LIN {X 0,Y 506.192,Z 351.476,A -85,B 0,C 180,E1 -5678.842,E2 -5678.842} C_VEL
LIN {X 0,Y 505.573,Z 365.781,A -85,B 0,C 180,E1 -5679.704,E2 -5679.704} C_VEL
LIN {X 0,Y 505.041,Z 378.228,A -85,B 0,C 180,E1 -5680.625,E2 -5680.625} C_VEL
LIN {X 0,Y 504.462,Z 389.865,A -85,B 0,C 180,E1 -5681.655,E2 -5681.655} C_VEL
LIN {X 0,Y 503.901,Z 401.554,A -85,B 0,C 180,E1 -5682.894,E2 -5682.894} C_VEL
LIN {X 0,Y 503.396,Z 411.462,A -85,B 0,C 180,E1 -5684.142,E2 -5684.142} C_VEL
LIN {X 0,Y 502.965,Z 421.023,A -85,B 0,C 180,E1 -5685.583,E2 -5685.583} C_VEL
LIN {X 0,Y 502.631,Z 429.216,A -85,B 0,C 180,E1 -5687.075,E2 -5687.075} C_VEL
LIN {X 0,Y 502.473,Z 434.837,A -85,B 0,C 180,E1 -5688.301,E2 -5688.301} C_VEL
LIN {X 0,Y 502.272,Z 441.149,A -85,B 0,C 180,E1 -5689.99,E2 -5689.99} C_VEL
LIN {X 0,Y 502.192,Z 445.104,A -85,B 0,C 180,E1 -5691.338,E2 -5691.338} C_VEL
LIN {X 0,Y 502.044,Z 448.907,A -85,B 0,C 180,E1 -5693.077,E2 -5693.077} C_VEL
LIN {X 0,Y 501.982,Z 451.304,A -85,B 0,C 180,E1 -5694.836,E2 -5694.836} C_VEL
LIN {X 0,Y 501.984,Z 452.341,A -85,B 0,C 180,E1 -5696.616,E2 -5696.616} C_VEL
LIN {X 0,Y 501.997,Z 451.979,A -85,B 0,C 180,E1 -5698.425,E2 -5698.425} C_VEL
LIN {X 0,Y 502.054,Z 450.118,A -85,B 0,C 180,E1 -5700.261,E2 -5700.261} C_VEL
LIN {X 0,Y 502.066,Z 448.297,A -85,B 0,C 180,E1 -5701.362,E2 -5701.362} C_VEL
LIN {X 0,Y 502.167,Z 444.274,A -85,B 0,C 180,E1 -5703.081,E2 -5703.081} C_VEL
LIN {X 0,Y 502.321,Z 439.329,A -85,B 0,C 180,E1 -5704.647,E2 -5704.647} C_VEL
LIN {X 0,Y 502.482,Z 433.012,A -85,B 0,C 180,E1 -5706.223,E2 -5706.223} C_VEL
LIN {X 0,Y 502.787,Z 425.506,A -85,B 0,C 180,E1 -5707.736,E2 -5707.736} C_VEL
LIN {X 0,Y 503.138,Z 416.684,A -85,B 0,C 180,E1 -5709.203,E2 -5709.203} C_VEL
LIN {X 0,Y 503.572,Z 407.62,A -85,B 0,C 180,E1 -5710.464,E2 -5710.464} C_VEL
LIN {X 0,Y 504.123,Z 396.604,A -85,B 0,C 180,E1 -5711.756,E2 -5711.756} C_VEL
LIN {X 0,Y 504.628,Z 385.523,A -85,B 0,C 180,E1 -5712.848,E2 -5712.848} C_VEL
LIN {X 0,Y 505.24,Z 373.889,A -85,B 0,C 180,E1 -5713.811,E2 -5713.811} C_VEL
LIN {X 0,Y 505.78,Z 361.268,A -85,B 0,C 180,E1 -5714.683,E2 -5714.683} C_VEL
LIN {X 0,Y 506.347,Z 346.906,A -85,B 0,C 180,E1 -5715.486,E2 -5715.486} C_VEL
LIN {X 0,Y 506.899,Z 331.848,A -85,B 0,C 180,E1 -5716.134,E2 -5716.134} C_VEL
LIN {X 0,Y 507.236,Z 316.604,A -85,B 0,C 180,E1 -5716.616,E2 -5716.616} C_VEL
LIN {X 0,Y 507.491,Z 300.362,A -85,B 0,C 180,E1 -5716.947,E2 -5716.947} C_VEL
LIN {X 0,Y 508.749,Z 153.983,A -85,B 0,C 180,E1 -5719.077,E2 -5719.077} C_VEL
LIN {X 0,Y 506.279,Z 139.939,A -85,B 0,C 180,E1 -5719.421,E2 -5719.421} C_VEL
LIN {X 0,Y 506.545,Z 123.358,A -85,B 0,C 180,E1 -5721.177,E2 -5721.177} C_VEL
LIN {X 0,Y 502.795,Z 108.482,A -85,B 0,C 180,E1 -5722.971,E2 -5722.971} C_VEL
LIN {X 0,Y 502.806,Z 108.482,A -85,B 0,C 180,E1 -5726.006,E2 -5726.006} C_VEL
LIN {X 0,Y 502.799,Z 108.477,A -85,B 0,C 180,E1 -5728.857,E2 -5728.857} C_VEL
LIN {X 0,Y 502.847,Z 108.477,A -85,B 0,C 180,E1 -5731.705,E2 -5731.705} C_VEL
LIN {X 0,Y 502.843,Z 108.473,A -85,B 0,C 180,E1 -5734.324,E2 -5734.324} C_VEL
LIN {X 0,Y 502.818,Z 108.529,A -85,B 0,C 180,E1 -5736.986,E2 -5736.986} C_VEL
LIN {X 0,Y 503.872,Z 112.951,A -85,B 0,C 180,E1 -5737.604,E2 -5737.604} C_VEL
LIN {X 0,Y 508.613,Z 125.414,A -85,B 0,C 180,E1 -5738.027,E2 -5738.027} C_VEL
LIN {X 0,Y 507.559,Z 222.564,A -85,B 0,C 180,E1 -5739.562,E2 -5739.562} C_VEL
LIN {X 0,Y 506.94,Z 279.945,A -85,B 0,C 180,E1 -5740.465,E2 -5740.465} C_VEL
LIN {X 0,Y 506.668,Z 295.372,A -85,B 0,C 180,E1 -5740.872,E2 -5740.872} C_VEL
LIN {X 0,Y 506.263,Z 310.367,A -85,B 0,C 180,E1 -5741.432,E2 -5741.432} C_VEL
LIN {X 0,Y 505.837,Z 324.005,A -85,B 0,C 180,E1 -5742.097,E2 -5742.097} C_VEL
LIN {X 0,Y 505.288,Z 337.428,A -85,B 0,C 180,E1 -5742.913,E2 -5742.913} C_VEL
LIN {X 0,Y 504.764,Z 350.501,A -85,B 0,C 180,E1 -5743.886,E2 -5743.886} C_VEL
LIN {X 0,Y 504.241,Z 363.457,A -85,B 0,C 180,E1 -5745.057,E2 -5745.057} C_VEL
LIN {X 0,Y 503.727,Z 374.703,A -85,B 0,C 180,E1 -5746.279,E2 -5746.279} C_VEL
LIN {X 0,Y 503.243,Z 385.732,A -85,B 0,C 180,E1 -5747.724,E2 -5747.724} C_VEL
LIN {X 0,Y 502.954,Z 394.624,A -85,B 0,C 180,E1 -5749.126,E2 -5749.126} C_VEL
LIN {X 0,Y 502.597,Z 403.052,A -85,B 0,C 180,E1 -5750.746,E2 -5750.746} C_VEL
LIN {X 0,Y 502.405,Z 409.809,A -85,B 0,C 180,E1 -5752.363,E2 -5752.363} C_VEL
LIN {X 0,Y 502.315,Z 415.092,A -85,B 0,C 180,E1 -5753.976,E2 -5753.976} C_VEL
LIN {X 0,Y 502.12,Z 418.131,A -85,B 0,C 180,E1 -5755.182,E2 -5755.182} C_VEL
LIN {X 0,Y 502.231,Z 421.123,A -85,B 0,C 180,E1 -5756.791,E2 -5756.791} C_VEL
LIN {X 0,Y 502.036,Z 422.952,A -85,B 0,C 180,E1 -5758.395,E2 -5758.395} C_VEL
LIN {X 0,Y 502.002,Z 423.613,A -85,B 0,C 180,E1 -5760,E2 -5760} C_VEL
LIN {X 0,Y 502.038,Z 423.077,A -85,B 0,C 180,E1 -5761.604,E2 -5761.604} C_VEL
LIN {X 0,Y 502.249,Z 421.385,A -85,B 0,C 180,E1 -5763.208,E2 -5763.208} C_VEL
LIN {X 0,Y 502.141,Z 418.525,A -85,B 0,C 180,E1 -5764.817,E2 -5764.817} C_VEL
LIN {X 0,Y 502.333,Z 414.388,A -85,B 0,C 180,E1 -5766.426,E2 -5766.426} C_VEL
LIN {X 0,Y 502.462,Z 408.89,A -85,B 0,C 180,E1 -5768.04,E2 -5768.04} C_VEL
LIN {X 0,Y 502.666,Z 401.854,A -85,B 0,C 180,E1 -5769.658,E2 -5769.658} C_VEL
LIN {X 0,Y 503.001,Z 394.271,A -85,B 0,C 180,E1 -5771.076,E2 -5771.076} C_VEL
LIN {X 0,Y 503.278,Z 385.393,A -85,B 0,C 180,E1 -5772.459,E2 -5772.459} C_VEL
LIN {X 0,Y 503.727,Z 375.704,A -85,B 0,C 180,E1 -5773.72,E2 -5773.72} C_VEL
LIN {X 0,Y 504.195,Z 364.498,A -85,B 0,C 180,E1 -5774.944,E2 -5774.944} C_VEL
LIN {X 0,Y 504.763,Z 351.596,A -85,B 0,C 180,E1 -5776.113,E2 -5776.113} C_VEL
LIN {X 0,Y 505.237,Z 338.543,A -85,B 0,C 180,E1 -5777.089,E2 -5777.089} C_VEL
LIN {X 0,Y 505.762,Z 325.103,A -85,B 0,C 180,E1 -5777.905,E2 -5777.905} C_VEL
LIN {X 0,Y 506.147,Z 311.424,A -85,B 0,C 180,E1 -5778.572,E2 -5778.572} C_VEL
LIN {X 0,Y 506.518,Z 296.117,A -85,B 0,C 180,E1 -5779.142,E2 -5779.142} C_VEL
LIN {X 0,Y 506.766,Z 280.632,A -85,B 0,C 180,E1 -5779.546,E2 -5779.546} C_VEL
LIN {X 0,Y 508.512,Z 155.31,A -85,B 0,C 180,E1 -5781.608,E2 -5781.608} C_VEL
LIN {X 0,Y 508.849,Z 129.1,A -85,B 0,C 180,E1 -5782.07,E2 -5782.07} C_VEL
LIN {X 0,Y 506.949,Z 122.35,A -85,B 0,C 180,E1 -5782.298,E2 -5782.298} C_VEL
LIN {X 0,Y 504.919,Z 117.566,A -85,B 0,C 180,E1 -5782.524,E2 -5782.524} C_VEL
LIN {X 0,Y 502.798,Z 108.482,A -85,B 0,C 180,E1 -5784.394,E2 -5784.394} C_VEL
LIN {X 0,Y 502.79,Z 108.484,A -85,B 0,C 180,E1 -5787.469,E2 -5787.469} C_VEL
LIN {X 0,Y 502.802,Z 108.48,A -85,B 0,C 180,E1 -5790.211,E2 -5790.211} C_VEL
LIN {X 0,Y 502.802,Z 108.48,A -85,B 0,C 180,E1 -5793.033,E2 -5793.033} C_VEL
LIN {X 0,Y 502.766,Z 108.485,A -85,B 0,C 180,E1 -5795.952,E2 -5795.952} C_VEL
LIN {X 0,Y 502.795,Z 108.481,A -85,B 0,C 180,E1 -5798.976,E2 -5798.976} C_VEL
LIN {X 0,Y 502.743,Z 108.484,A -85,B 0,C 180,E1 -5802.192,E2 -5802.192} C_VEL
LIN {X 0,Y 502.784,Z 108.483,A -85,B 0,C 180,E1 -5805.47,E2 -5805.47} C_VEL
LIN {X 0,Y 502.763,Z 108.487,A -85,B 0,C 180,E1 -5808.928,E2 -5808.928} C_VEL
LIN {X 0,Y 502.788,Z 108.479,A -85,B 0,C 180,E1 -5812.046,E2 -5812.046} C_VEL
LIN {X 0,Y 502.786,Z 108.485,A -85,B 0,C 180,E1 -5815.033,E2 -5815.033} C_VEL
LIN {X 0,Y 502.771,Z 108.484,A -85,B 0,C 180,E1 -5817.914,E2 -5817.914} C_VEL
LIN {X 0,Y 502.802,Z 108.672,A -85,B 0,C 180,E1 -5819.834,E2 -5819.834} C_VEL
LIN {X 0,Y 505.92,Z 121.058,A -85,B 0,C 180,E1 -5821.816,E2 -5821.816} C_VEL
LIN {X 0,Y 506.557,Z 124.311,A -85,B 0,C 180,E1 -5822.304,E2 -5822.304} C_VEL
LIN {X 0,Y 505.722,Z 144.394,A -85,B 0,C 180,E1 -5824.967,E2 -5824.967} C_VEL
LIN {X 0,Y 504.954,Z 164.114,A -85,B 0,C 180,E1 -5827.496,E2 -5827.496} C_VEL
LIN {X 0,Y 508.497,Z 185.654,A -85,B 0,C 180,E1 -5828.073,E2 -5828.073} C_VEL
LIN {X 0,Y 507.022,Z 292.758,A -85,B 0,C 180,E1 -5829.83,E2 -5829.83} C_VEL
LIN {X 0,Y 506.548,Z 333.914,A -85,B 0,C 180,E1 -5830.497,E2 -5830.497} C_VEL
LIN {X 0,Y 506.136,Z 349.417,A -85,B 0,C 180,E1 -5830.905,E2 -5830.905} C_VEL
LIN {X 0,Y 505.713,Z 364.455,A -85,B 0,C 180,E1 -5831.464,E2 -5831.464} C_VEL
LIN {X 0,Y 505.165,Z 379.158,A -85,B 0,C 180,E1 -5832.177,E2 -5832.177} C_VEL
LIN {X 0,Y 504.657,Z 392.632,A -85,B 0,C 180,E1 -5832.995,E2 -5832.995} C_VEL
LIN {X 0,Y 504.186,Z 406.022,A -85,B 0,C 180,E1 -5833.987,E2 -5833.987} C_VEL
LIN {X 0,Y 503.687,Z 417.91,A -85,B 0,C 180,E1 -5835.041,E2 -5835.041} C_VEL
LIN {X 0,Y 503.287,Z 429.5,A -85,B 0,C 180,E1 -5836.267,E2 -5836.267} C_VEL
LIN {X 0,Y 502.932,Z 439.231,A -85,B 0,C 180,E1 -5837.491,E2 -5837.491} C_VEL
LIN {X 0,Y 502.691,Z 447.494,A -85,B 0,C 180,E1 -5838.713,E2 -5838.713} C_VEL
LIN {X 0,Y 502.423,Z 455.624,A -85,B 0,C 180,E1 -5840.133,E2 -5840.133} C_VEL
LIN {X 0,Y 502.285,Z 462.353,A -85,B 0,C 180,E1 -5841.552,E2 -5841.552} C_VEL
LIN {X 0,Y 502.221,Z 468.522,A -85,B 0,C 180,E1 -5843.169,E2 -5843.169} C_VEL
LIN {X 0,Y 502.146,Z 473.251,A -85,B 0,C 180,E1 -5844.78,E2 -5844.78} C_VEL
LIN {X 0,Y 502.13,Z 475.867,A -85,B 0,C 180,E1 -5845.987,E2 -5845.987} C_VEL
LIN {X 0,Y 502.117,Z 478.31,A -85,B 0,C 180,E1 -5847.593,E2 -5847.593} C_VEL
LIN {X 0,Y 501.993,Z 479.548,A -85,B 0,C 180,E1 -5849.198,E2 -5849.198} C_VEL
LIN {X 0,Y 501.992,Z 479.577,A -85,B 0,C 180,E1 -5850.802,E2 -5850.802} C_VEL
LIN {X 0,Y 502.117,Z 478.396,A -85,B 0,C 180,E1 -5852.407,E2 -5852.407} C_VEL
LIN {X 0,Y 502.129,Z 476.018,A -85,B 0,C 180,E1 -5854.013,E2 -5854.013} C_VEL
LIN {X 0,Y 502.195,Z 472.398,A -85,B 0,C 180,E1 -5855.622,E2 -5855.622} C_VEL
LIN {X 0,Y 502.234,Z 467.436,A -85,B 0,C 180,E1 -5857.235,E2 -5857.235} C_VEL
LIN {X 0,Y 502.313,Z 461,A -85,B 0,C 180,E1 -5858.853,E2 -5858.853} C_VEL
LIN {X 0,Y 502.584,Z 452.92,A -85,B 0,C 180,E1 -5860.474,E2 -5860.474} C_VEL
LIN {X 0,Y 502.804,Z 444.129,A -85,B 0,C 180,E1 -5861.922,E2 -5861.922} C_VEL
LIN {X 0,Y 503.195,Z 433.884,A -85,B 0,C 180,E1 -5863.324,E2 -5863.324} C_VEL
LIN {X 0,Y 503.616,Z 423.234,A -85,B 0,C 180,E1 -5864.548,E2 -5864.548} C_VEL
LIN {X 0,Y 504.109,Z 410.905,A -85,B 0,C 180,E1 -5865.736,E2 -5865.736} C_VEL
LIN {X 0,Y 504.603,Z 399.061,A -85,B 0,C 180,E1 -5866.694,E2 -5866.694} C_VEL
LIN {X 0,Y 505.206,Z 385.293,A -85,B 0,C 180,E1 -5867.612,E2 -5867.612} C_VEL
LIN {X 0,Y 505.75,Z 371.064,A -85,B 0,C 180,E1 -5868.377,E2 -5868.377} C_VEL
LIN {X 0,Y 506.262,Z 356.646,A -85,B 0,C 180,E1 -5868.982,E2 -5868.982} C_VEL
LIN {X 0,Y 506.665,Z 341.674,A -85,B 0,C 180,E1 -5869.445,E2 -5869.445} C_VEL
LIN {X 0,Y 506.929,Z 325.194,A -85,B 0,C 180,E1 -5869.777,E2 -5869.777} C_VEL
LIN {X 0,Y 508.535,Z 184.49,A -85,B 0,C 180,E1 -5871.962,E2 -5871.962} C_VEL
LIN {X 0,Y 508.192,Z 179.447,A -85,B 0,C 180,E1 -5872.061,E2 -5872.061} C_VEL
LIN {X 0,Y 506.015,Z 165.025,A -85,B 0,C 180,E1 -5872.411,E2 -5872.411} C_VEL
LIN {X 0,Y 506.86,Z 142.117,A -85,B 0,C 180,E1 -5874.69,E2 -5874.69} C_VEL
LIN {X 0,Y 507.529,Z 126.06,A -85,B 0,C 180,E1 -5876.303,E2 -5876.303} C_VEL
LIN {X 0,Y 502.788,Z 108.483,A -85,B 0,C 180,E1 -5878.404,E2 -5878.404} C_VEL
LIN {X 0,Y 502.785,Z 108.484,A -85,B 0,C 180,E1 -5881.144,E2 -5881.144} C_VEL
LIN {X 0,Y 502.785,Z 108.478,A -85,B 0,C 180,E1 -5883.995,E2 -5883.995} C_VEL
LIN {X 0,Y 502.763,Z 108.486,A -85,B 0,C 180,E1 -5887.176,E2 -5887.176} C_VEL
LIN {X 0,Y 502.77,Z 108.481,A -85,B 0,C 180,E1 -5890.017,E2 -5890.017} C_VEL
LIN {X 0,Y 502.746,Z 108.484,A -85,B 0,C 180,E1 -5893.234,E2 -5893.234} C_VEL
LIN {X 0,Y 502.777,Z 108.476,A -85,B 0,C 180,E1 -5895.66,E2 -5895.66} C_VEL
LIN {X 0,Y 502.764,Z 108.483,A -85,B 0,C 180,E1 -5899.012,E2 -5899.012} C_VEL
LIN {X 0,Y 502.789,Z 108.48,A -85,B 0,C 180,E1 -5902.046,E2 -5902.046} C_VEL
LIN {X 0,Y 502.791,Z 108.48,A -85,B 0,C 180,E1 -5905.034,E2 -5905.034} C_VEL
LIN {X 0,Y 502.781,Z 108.482,A -85,B 0,C 180,E1 -5907.915,E2 -5907.915} C_VEL
LIN {X 0,Y 502.804,Z 108.481,A -85,B 0,C 180,E1 -5910.711,E2 -5910.711} C_VEL
LIN {X 0,Y 502.774,Z 108.482,A -85,B 0,C 180,E1 -5913.46,E2 -5913.46} C_VEL
LIN {X 0,Y 502.786,Z 108.557,A -85,B 0,C 180,E1 -5916.387,E2 -5916.387} C_VEL
LIN {X 0,Y 504.707,Z 116.182,A -85,B 0,C 180,E1 -5917.588,E2 -5917.588} C_VEL
LIN {X 0,Y 507.891,Z 125.008,A -85,B 0,C 180,E1 -5917.921,E2 -5917.921} C_VEL
LIN {X 0,Y 508.835,Z 129.707,A -85,B 0,C 180,E1 -5918.056,E2 -5918.056} C_VEL
LIN {X 0,Y 507.257,Z 231.397,A -85,B 0,C 180,E1 -5919.761,E2 -5919.761} C_VEL
LIN {X 0,Y 506.727,Z 280.59,A -85,B 0,C 180,E1 -5920.557,E2 -5920.557} C_VEL
LIN {X 0,Y 506.476,Z 295.923,A -85,B 0,C 180,E1 -5920.956,E2 -5920.956} C_VEL
LIN {X 0,Y 506.123,Z 310.178,A -85,B 0,C 180,E1 -5921.48,E2 -5921.48} C_VEL
LIN {X 0,Y 505.757,Z 323.108,A -85,B 0,C 180,E1 -5922.095,E2 -5922.095} C_VEL
LIN {X 0,Y 505.238,Z 336.924,A -85,B 0,C 180,E1 -5922.911,E2 -5922.911} C_VEL
LIN {X 0,Y 504.732,Z 350.42,A -85,B 0,C 180,E1 -5923.898,E2 -5923.898} C_VEL
LIN {X 0,Y 504.25,Z 362.346,A -85,B 0,C 180,E1 -5924.955,E2 -5924.955} C_VEL
LIN {X 0,Y 503.807,Z 373.008,A -85,B 0,C 180,E1 -5926.076,E2 -5926.076} C_VEL
LIN {X 0,Y 503.419,Z 382.834,A -85,B 0,C 180,E1 -5927.299,E2 -5927.299} C_VEL
LIN {X 0,Y 503.038,Z 392.387,A -85,B 0,C 180,E1 -5928.721,E2 -5928.721} C_VEL
LIN {X 0,Y 502.689,Z 400.304,A -85,B 0,C 180,E1 -5930.139,E2 -5930.139} C_VEL
LIN {X 0,Y 502.515,Z 406.842,A -85,B 0,C 180,E1 -5931.556,E2 -5931.556} C_VEL
LIN {X 0,Y 502.311,Z 412.936,A -85,B 0,C 180,E1 -5933.21,E2 -5933.21} C_VEL
LIN {X 0,Y 502.275,Z 416.298,A -85,B 0,C 180,E1 -5934.379,E2 -5934.379} C_VEL
LIN {X 0,Y 502.189,Z 419.867,A -85,B 0,C 180,E1 -5935.988,E2 -5935.988} C_VEL
LIN {X 0,Y 502.13,Z 422.215,A -85,B 0,C 180,E1 -5937.594,E2 -5937.594} C_VEL
LIN {X 0,Y 502.003,Z 423.399,A -85,B 0,C 180,E1 -5939.198,E2 -5939.198} C_VEL
LIN {X 0,Y 502.003,Z 423.386,A -85,B 0,C 180,E1 -5940.802,E2 -5940.802} C_VEL
LIN {X 0,Y 502.131,Z 422.213,A -85,B 0,C 180,E1 -5942.407,E2 -5942.407} C_VEL
LIN {X 0,Y 502.188,Z 419.88,A -85,B 0,C 180,E1 -5944.013,E2 -5944.013} C_VEL
LIN {X 0,Y 502.267,Z 416.329,A -85,B 0,C 180,E1 -5945.621,E2 -5945.621} C_VEL
LIN {X 0,Y 502.361,Z 411.477,A -85,B 0,C 180,E1 -5947.234,E2 -5947.234} C_VEL
LIN {X 0,Y 502.508,Z 405.194,A -85,B 0,C 180,E1 -5948.85,E2 -5948.85} C_VEL
LIN {X 0,Y 502.772,Z 397.283,A -85,B 0,C 180,E1 -5950.47,E2 -5950.47} C_VEL
LIN {X 0,Y 503.038,Z 388.849,A -85,B 0,C 180,E1 -5951.887,E2 -5951.887} C_VEL
LIN {X 0,Y 503.54,Z 378.594,A -85,B 0,C 180,E1 -5953.315,E2 -5953.315} C_VEL
LIN {X 0,Y 504.008,Z 368.103,A -85,B 0,C 180,E1 -5954.537,E2 -5954.537} C_VEL
LIN {X 0,Y 504.5,Z 356.654,A -85,B 0,C 180,E1 -5955.66,E2 -5955.66} C_VEL
LIN {X 0,Y 505.013,Z 344.225,A -85,B 0,C 180,E1 -5956.68,E2 -5956.68} C_VEL
LIN {X 0,Y 505.543,Z 330.609,A -85,B 0,C 180,E1 -5957.6,E2 -5957.6} C_VEL
LIN {X 0,Y 506.037,Z 316.494,A -85,B 0,C 180,E1 -5958.367,E2 -5958.367} C_VEL
LIN {X 0,Y 506.511,Z 300.879,A -85,B 0,C 180,E1 -5959.02,E2 -5959.02} C_VEL
LIN {X 0,Y 506.843,Z 285.314,A -85,B 0,C 180,E1 -5959.491,E2 -5959.491} C_VEL
LIN {X 0,Y 507.044,Z 269.676,A -85,B 0,C 180,E1 -5959.799,E2 -5959.799} C_VEL
LIN {X 0,Y 508.646,Z 129.723,A -85,B 0,C 180,E1 -5961.977,E2 -5961.977} C_VEL
LIN {X 0,Y 506.606,Z 120.903,A -85,B 0,C 180,E1 -5962.212,E2 -5962.212} C_VEL
LIN {X 0,Y 503.925,Z 113.653,A -85,B 0,C 180,E1 -5962.479,E2 -5962.479} C_VEL
LIN {X 0,Y 502.805,Z 108.48,A -85,B 0,C 180,E1 -5963.367,E2 -5963.367} C_VEL
LIN {X 0,Y 502.814,Z 108.475,A -85,B 0,C 180,E1 -5966.569,E2 -5966.569} C_VEL
LIN {X 0,Y 502.812,Z 108.48,A -85,B 0,C 180,E1 -5969.934,E2 -5969.934} C_VEL
LIN {X 0,Y 502.804,Z 108.477,A -85,B 0,C 180,E1 -5973.034,E2 -5973.034} C_VEL
LIN {X 0,Y 502.77,Z 108.483,A -85,B 0,C 180,E1 -5975.888,E2 -5975.888} C_VEL
LIN {X 0,Y 502.096,Z 108.564,A -85,B 0,C 180,E1 -5976.556,E2 -5976.556} C_VEL
LIN {X 0,Y 499.241,Z 108.925,A -85,B 0,C 180,E1 -5977.64,E2 -5977.64} C_VEL
LIN {X 0,Y 496.837,Z 109.22,A -85,B 0,C 180,E1 -5978.514,E2 -5978.514} C_VEL
LIN {X 0,Y 495.816,Z 109.349,A -85,B 0,C 180,E1 -5979.189,E2 -5979.189} C_VEL
LIN {X 0,Y 495.738,Z 109.358,A -85,B 0,C 180,E1 -5979.417,E2 -5979.417} C_VEL
LIN {X 0,Y 495.714,Z 109.358,A -85,B 0,C 180,E1 -5982.504,E2 -5982.504} C_VEL
LIN {X 0,Y 495.739,Z 109.355,A -85,B 0,C 180,E1 -5985.141,E2 -5985.141} C_VEL
LIN {X 0,Y 495.726,Z 109.351,A -85,B 0,C 180,E1 -5988.216,E2 -5988.216} C_VEL
LIN {X 0,Y 495.748,Z 109.357,A -85,B 0,C 180,E1 -5991.408,E2 -5991.408} C_VEL
LIN {X 0,Y 495.745,Z 109.346,A -85,B 0,C 180,E1 -5994.462,E2 -5994.462} C_VEL
LIN {X 0,Y 495.753,Z 109.356,A -85,B 0,C 180,E1 -5997.404,E2 -5997.404} C_VEL
LIN {X 0,Y 495.742,Z 109.35,A -85,B 0,C 180,E1 -6000.252,E2 -6000.252} C_VEL
LIN {X 0,Y 495.742,Z 109.357,A -85,B 0,C 180,E1 -6003.271,E2 -6003.271} C_VEL
LIN {X 0,Y 495.737,Z 109.355,A -85,B 0,C 180,E1 -6006.612,E2 -6006.612} C_VEL
LIN {X 0,Y 495.782,Z 109.348,A -85,B 0,C 180,E1 -6009.324,E2 -6009.324} C_VEL
LIN {X 0,Y 495.764,Z 109.352,A -85,B 0,C 180,E1 -6011.828,E2 -6011.828} C_VEL
LIN {X 0,Y 495.777,Z 109.352,A -85,B 0,C 180,E1 -6015.217,E2 -6015.217} C_VEL
LIN {X 0,Y 495.854,Z 109.346,A -85,B 0,C 180,E1 -6018.555,E2 -6018.555} C_VEL
LIN {X 0,Y 495.814,Z 109.348,A -85,B 0,C 180,E1 -6021.851,E2 -6021.851} C_VEL
LIN {X 0,Y 495.819,Z 109.347,A -85,B 0,C 180,E1 -6025.121,E2 -6025.121} C_VEL
LIN {X 0,Y 495.977,Z 109.33,A -85,B 0,C 180,E1 -6027.564,E2 -6027.564} C_VEL
LIN {X 0,Y 495.904,Z 109.404,A -85,B 0,C 180,E1 -6029.746,E2 -6029.746} C_VEL
LIN {X 0,Y 498.874,Z 123.212,A -85,B 0,C 180,E1 -6031.816,E2 -6031.816} C_VEL
LIN {X 0,Y 498.743,Z 134.952,A -85,B 0,C 180,E1 -6033.433,E2 -6033.433} C_VEL
LIN {X 0,Y 498.575,Z 141.915,A -85,B 0,C 180,E1 -6034.36,E2 -6034.36} C_VEL
LIN {X 0,Y 502.108,Z 158.195,A -85,B 0,C 180,E1 -6034.776,E2 -6034.776} C_VEL
LIN {X 0,Y 500.735,Z 307.945,A -85,B 0,C 180,E1 -6037.004,E2 -6037.004} C_VEL
LIN {X 0,Y 500.429,Z 323.034,A -85,B 0,C 180,E1 -6037.388,E2 -6037.388} C_VEL
LIN {X 0,Y 499.964,Z 337.824,A -85,B 0,C 180,E1 -6037.928,E2 -6037.928} C_VEL
LIN {X 0,Y 499.425,Z 351.76,A -85,B 0,C 180,E1 -6038.599,E2 -6038.599} C_VEL
LIN {X 0,Y 498.832,Z 364.756,A -85,B 0,C 180,E1 -6039.381,E2 -6039.381} C_VEL
LIN {X 0,Y 498.254,Z 377.945,A -85,B 0,C 180,E1 -6040.361,E2 -6040.361} C_VEL
LIN {X 0,Y 497.581,Z 389.69,A -85,B 0,C 180,E1 -6041.405,E2 -6041.405} C_VEL
LIN {X 0,Y 496.995,Z 401.325,A -85,B 0,C 180,E1 -6042.648,E2 -6042.648} C_VEL
LIN {X 0,Y 496.464,Z 411.384,A -85,B 0,C 180,E1 -6043.925,E2 -6043.925} C_VEL
LIN {X 0,Y 495.961,Z 420.964,A -85,B 0,C 180,E1 -6045.381,E2 -6045.381} C_VEL
LIN {X 0,Y 495.606,Z 429.237,A -85,B 0,C 180,E1 -6046.9,E2 -6046.9} C_VEL
LIN {X 0,Y 495.439,Z 435.041,A -85,B 0,C 180,E1 -6048.185,E2 -6048.185} C_VEL
LIN {X 0,Y 495.213,Z 441.414,A -85,B 0,C 180,E1 -6049.914,E2 -6049.914} C_VEL
LIN {X 0,Y 495.073,Z 446.303,A -85,B 0,C 180,E1 -6051.66,E2 -6051.66} C_VEL
LIN {X 0,Y 494.924,Z 449.786,A -85,B 0,C 180,E1 -6053.429,E2 -6053.429} C_VEL
LIN {X 0,Y 494.866,Z 451.874,A -85,B 0,C 180,E1 -6055.217,E2 -6055.217} C_VEL
LIN {X 0,Y 494.886,Z 452.604,A -85,B 0,C 180,E1 -6057.029,E2 -6057.029} C_VEL
LIN {X 0,Y 494.914,Z 451.885,A -85,B 0,C 180,E1 -6058.869,E2 -6058.869} C_VEL
LIN {X 0,Y 494.954,Z 450.732,A -85,B 0,C 180,E1 -6059.984,E2 -6059.984} C_VEL
LIN {X 0,Y 495,Z 447.939,A -85,B 0,C 180,E1 -6061.69,E2 -6061.69} C_VEL
LIN {X 0,Y 495.089,Z 444.599,A -85,B 0,C 180,E1 -6063.119,E2 -6063.119} C_VEL
LIN {X 0,Y 495.238,Z 440.025,A -85,B 0,C 180,E1 -6064.604,E2 -6064.604} C_VEL
LIN {X 0,Y 495.425,Z 433.546,A -85,B 0,C 180,E1 -6066.27,E2 -6066.27} C_VEL
LIN {X 0,Y 495.763,Z 426.061,A -85,B 0,C 180,E1 -6067.815,E2 -6067.815} C_VEL
LIN {X 0,Y 496.148,Z 416.844,A -85,B 0,C 180,E1 -6069.379,E2 -6069.379} C_VEL
LIN {X 0,Y 496.627,Z 408.089,A -85,B 0,C 180,E1 -6070.615,E2 -6070.615} C_VEL
LIN {X 0,Y 497.193,Z 397.305,A -85,B 0,C 180,E1 -6071.905,E2 -6071.905} C_VEL
LIN {X 0,Y 497.73,Z 386.135,A -85,B 0,C 180,E1 -6073.029,E2 -6073.029} C_VEL
LIN {X 0,Y 498.398,Z 374.453,A -85,B 0,C 180,E1 -6074.014,E2 -6074.014} C_VEL
LIN {X 0,Y 498.967,Z 361.909,A -85,B 0,C 180,E1 -6074.899,E2 -6074.899} C_VEL
LIN {X 0,Y 499.556,Z 348.544,A -85,B 0,C 180,E1 -6075.667,E2 -6075.667} C_VEL
LIN {X 0,Y 500.071,Z 334.693,A -85,B 0,C 180,E1 -6076.297,E2 -6076.297} C_VEL
LIN {X 0,Y 500.485,Z 319.626,A -85,B 0,C 180,E1 -6076.808,E2 -6076.808} C_VEL
LIN {X 0,Y 500.776,Z 304.499,A -85,B 0,C 180,E1 -6077.154,E2 -6077.154} C_VEL
LIN {X 0,Y 502.12,Z 154.7,A -85,B 0,C 180,E1 -6079.375,E2 -6079.375} C_VEL
LIN {X 0,Y 499.566,Z 140.129,A -85,B 0,C 180,E1 -6079.739,E2 -6079.739} C_VEL
LIN {X 0,Y 499.82,Z 125.746,A -85,B 0,C 180,E1 -6081.265,E2 -6081.265} C_VEL
LIN {X 0,Y 496.736,Z 113.065,A -85,B 0,C 180,E1 -6082.782,E2 -6082.782} C_VEL
LIN {X 0,Y 495.738,Z 109.361,A -85,B 0,C 180,E1 -6083.235,E2 -6083.235} C_VEL
LIN {X 0,Y 495.762,Z 109.356,A -85,B 0,C 180,E1 -6086.435,E2 -6086.435} C_VEL
LIN {X 0,Y 495.754,Z 109.357,A -85,B 0,C 180,E1 -6089.313,E2 -6089.313} C_VEL
LIN {X 0,Y 495.783,Z 109.353,A -85,B 0,C 180,E1 -6092.109,E2 -6092.109} C_VEL
LIN {X 0,Y 495.791,Z 109.353,A -85,B 0,C 180,E1 -6094.833,E2 -6094.833} C_VEL
LIN {X 0,Y 495.786,Z 109.479,A -85,B 0,C 180,E1 -6096.738,E2 -6096.738} C_VEL
LIN {X 0,Y 496.666,Z 113.123,A -85,B 0,C 180,E1 -6097.266,E2 -6097.266} C_VEL
LIN {X 0,Y 502.103,Z 127.448,A -85,B 0,C 180,E1 -6097.765,E2 -6097.765} C_VEL
LIN {X 0,Y 500.205,Z 279.83,A -85,B 0,C 180,E1 -6100.213,E2 -6100.213} C_VEL
LIN {X 0,Y 499.902,Z 295.651,A -85,B 0,C 180,E1 -6100.634,E2 -6100.634} C_VEL
LIN {X 0,Y 499.443,Z 311.103,A -85,B 0,C 180,E1 -6101.222,E2 -6101.222} C_VEL
LIN {X 0,Y 498.961,Z 325.553,A -85,B 0,C 180,E1 -6101.948,E2 -6101.948} C_VEL
LIN {X 0,Y 498.39,Z 338.785,A -85,B 0,C 180,E1 -6102.774,E2 -6102.774} C_VEL
LIN {X 0,Y 497.87,Z 351.208,A -85,B 0,C 180,E1 -6103.719,E2 -6103.719} C_VEL
LIN {X 0,Y 497.344,Z 363.501,A -85,B 0,C 180,E1 -6104.845,E2 -6104.845} C_VEL
LIN {X 0,Y 496.786,Z 374.813,A -85,B 0,C 180,E1 -6106.084,E2 -6106.084} C_VEL
LIN {X 0,Y 496.272,Z 385.775,A -85,B 0,C 180,E1 -6107.528,E2 -6107.528} C_VEL
LIN {X 0,Y 495.953,Z 394.846,A -85,B 0,C 180,E1 -6108.971,E2 -6108.971} C_VEL
LIN {X 0,Y 495.559,Z 403.319,A -85,B 0,C 180,E1 -6110.613,E2 -6110.613} C_VEL
LIN {X 0,Y 495.344,Z 410.112,A -85,B 0,C 180,E1 -6112.253,E2 -6112.253} C_VEL
LIN {X 0,Y 495.219,Z 414.854,A -85,B 0,C 180,E1 -6113.694,E2 -6113.694} C_VEL
LIN {X 0,Y 495.046,Z 418.482,A -85,B 0,C 180,E1 -6115.113,E2 -6115.113} C_VEL
LIN {X 0,Y 495.143,Z 421.494,A -85,B 0,C 180,E1 -6116.745,E2 -6116.745} C_VEL
LIN {X 0,Y 494.963,Z 423.34,A -85,B 0,C 180,E1 -6118.372,E2 -6118.372} C_VEL
LIN {X 0,Y 494.918,Z 424.01,A -85,B 0,C 180,E1 -6120,E2 -6120} C_VEL
LIN {X 0,Y 494.965,Z 423.477,A -85,B 0,C 180,E1 -6121.627,E2 -6121.627} C_VEL
LIN {X 0,Y 495.159,Z 421.781,A -85,B 0,C 180,E1 -6123.254,E2 -6123.254} C_VEL
LIN {X 0,Y 495.067,Z 418.907,A -85,B 0,C 180,E1 -6124.886,E2 -6124.886} C_VEL
LIN {X 0,Y 495.291,Z 414.751,A -85,B 0,C 180,E1 -6126.518,E2 -6126.518} C_VEL
LIN {X 0,Y 495.426,Z 409.229,A -85,B 0,C 180,E1 -6128.155,E2 -6128.155} C_VEL
LIN {X 0,Y 495.637,Z 402.165,A -85,B 0,C 180,E1 -6129.797,E2 -6129.797} C_VEL
LIN {X 0,Y 495.988,Z 394.542,A -85,B 0,C 180,E1 -6131.235,E2 -6131.235} C_VEL
LIN {X 0,Y 496.317,Z 385.325,A -85,B 0,C 180,E1 -6132.679,E2 -6132.679} C_VEL
LIN {X 0,Y 496.789,Z 375.909,A -85,B 0,C 180,E1 -6133.916,E2 -6133.916} C_VEL
LIN {X 0,Y 497.303,Z 364.661,A -85,B 0,C 180,E1 -6135.156,E2 -6135.156} C_VEL
LIN {X 0,Y 497.887,Z 352.333,A -85,B 0,C 180,E1 -6136.288,E2 -6136.288} C_VEL
LIN {X 0,Y 498.366,Z 340.064,A -85,B 0,C 180,E1 -6137.226,E2 -6137.226} C_VEL
LIN {X 0,Y 498.91,Z 326.871,A -85,B 0,C 180,E1 -6138.053,E2 -6138.053} C_VEL
LIN {X 0,Y 499.3,Z 313.54,A -85,B 0,C 180,E1 -6138.729,E2 -6138.729} C_VEL
LIN {X 0,Y 499.711,Z 298.98,A -85,B 0,C 180,E1 -6139.302,E2 -6139.302} C_VEL
LIN {X 0,Y 499.953,Z 283.457,A -85,B 0,C 180,E1 -6139.744,E2 -6139.744} C_VEL
LIN {X 0,Y 500.391,Z 251.828,A -85,B 0,C 180,E1 -6140.288,E2 -6140.288} C_VEL
LIN {X 0,Y 502.015,Z 154.428,A -85,B 0,C 180,E1 -6141.949,E2 -6141.949} C_VEL
LIN {X 0,Y 502.379,Z 130.346,A -85,B 0,C 180,E1 -6142.392,E2 -6142.392} C_VEL
LIN {X 0,Y 500.711,Z 124.909,A -85,B 0,C 180,E1 -6142.586,E2 -6142.586} C_VEL
LIN {X 0,Y 497.922,Z 118.309,A -85,B 0,C 180,E1 -6142.902,E2 -6142.902} C_VEL
LIN {X 0,Y 495.733,Z 109.361,A -85,B 0,C 180,E1 -6144.828,E2 -6144.828} C_VEL
LIN {X 0,Y 495.755,Z 109.359,A -85,B 0,C 180,E1 -6146.977,E2 -6146.977} C_VEL
LIN {X 0,Y 495.758,Z 109.358,A -85,B 0,C 180,E1 -6150.146,E2 -6150.146} C_VEL
LIN {X 0,Y 495.751,Z 109.359,A -85,B 0,C 180,E1 -6153.237,E2 -6153.237} C_VEL
LIN {X 0,Y 495.71,Z 109.362,A -85,B 0,C 180,E1 -6156.087,E2 -6156.087} C_VEL
LIN {X 0,Y 495.758,Z 109.356,A -85,B 0,C 180,E1 -6158.767,E2 -6158.767} C_VEL
LIN {X 0,Y 495.722,Z 109.362,A -85,B 0,C 180,E1 -6161.784,E2 -6161.784} C_VEL
LIN {X 0,Y 495.736,Z 109.361,A -85,B 0,C 180,E1 -6165.141,E2 -6165.141} C_VEL
LIN {X 0,Y 495.722,Z 109.359,A -85,B 0,C 180,E1 -6168.215,E2 -6168.215} C_VEL
LIN {X 0,Y 495.744,Z 109.361,A -85,B 0,C 180,E1 -6171.408,E2 -6171.408} C_VEL
LIN {X 0,Y 495.738,Z 109.362,A -85,B 0,C 180,E1 -6174.461,E2 -6174.461} C_VEL
LIN {X 0,Y 495.747,Z 109.36,A -85,B 0,C 180,E1 -6177.404,E2 -6177.404} C_VEL
LIN {X 0,Y 495.74,Z 109.519,A -85,B 0,C 180,E1 -6179.427,E2 -6179.427} C_VEL
LIN {X 0,Y 499.149,Z 122.777,A -85,B 0,C 180,E1 -6181.628,E2 -6181.628} C_VEL
LIN {X 0,Y 499.783,Z 125.95,A -85,B 0,C 180,E1 -6182.124,E2 -6182.124} C_VEL
LIN {X 0,Y 498.979,Z 144.757,A -85,B 0,C 180,E1 -6184.674,E2 -6184.674} C_VEL
LIN {X 0,Y 498.143,Z 163.672,A -85,B 0,C 180,E1 -6187.137,E2 -6187.137} C_VEL
LIN {X 0,Y 501.609,Z 184.596,A -85,B 0,C 180,E1 -6187.718,E2 -6187.718} C_VEL
LIN {X 0,Y 501.916,Z 187.381,A -85,B 0,C 180,E1 -6187.786,E2 -6187.786} C_VEL
LIN {X 0,Y 500.31,Z 292.945,A -85,B 0,C 180,E1 -6189.575,E2 -6189.575} C_VEL
LIN {X 0,Y 499.762,Z 333.443,A -85,B 0,C 180,E1 -6190.248,E2 -6190.248} C_VEL
LIN {X 0,Y 499.341,Z 349.207,A -85,B 0,C 180,E1 -6190.674,E2 -6190.674} C_VEL
LIN {X 0,Y 498.857,Z 364.422,A -85,B 0,C 180,E1 -6191.253,E2 -6191.253} C_VEL
LIN {X 0,Y 498.303,Z 378.101,A -85,B 0,C 180,E1 -6191.924,E2 -6191.924} C_VEL
LIN {X 0,Y 497.693,Z 393.187,A -85,B 0,C 180,E1 -6192.856,E2 -6192.856} C_VEL
LIN {X 0,Y 497.163,Z 407.044,A -85,B 0,C 180,E1 -6193.914,E2 -6193.914} C_VEL
LIN {X 0,Y 496.649,Z 419.178,A -85,B 0,C 180,E1 -6195.034,E2 -6195.034} C_VEL
LIN {X 0,Y 496.206,Z 430.469,A -85,B 0,C 180,E1 -6196.276,E2 -6196.276} C_VEL
LIN {X 0,Y 495.857,Z 440.047,A -85,B 0,C 180,E1 -6197.517,E2 -6197.517} C_VEL
LIN {X 0,Y 495.539,Z 449.401,A -85,B 0,C 180,E1 -6198.962,E2 -6198.962} C_VEL
LIN {X 0,Y 495.289,Z 457.158,A -85,B 0,C 180,E1 -6200.402,E2 -6200.402} C_VEL
LIN {X 0,Y 495.196,Z 463.519,A -85,B 0,C 180,E1 -6201.841,E2 -6201.841} C_VEL
LIN {X 0,Y 495.091,Z 469.568,A -85,B 0,C 180,E1 -6203.552,E2 -6203.552} C_VEL
LIN {X 0,Y 495.01,Z 473.732,A -85,B 0,C 180,E1 -6205.113,E2 -6205.113} C_VEL
LIN {X 0,Y 495.031,Z 476.822,A -85,B 0,C 180,E1 -6206.745,E2 -6206.745} C_VEL
LIN {X 0,Y 494.96,Z 478.672,A -85,B 0,C 180,E1 -6208.373,E2 -6208.373} C_VEL
LIN {X 0,Y 494.908,Z 479.327,A -85,B 0,C 180,E1 -6210,E2 -6210} C_VEL
LIN {X 0,Y 494.96,Z 478.742,A -85,B 0,C 180,E1 -6211.627,E2 -6211.627} C_VEL
LIN {X 0,Y 495.031,Z 476.962,A -85,B 0,C 180,E1 -6213.255,E2 -6213.255} C_VEL
LIN {X 0,Y 495.006,Z 473.956,A -85,B 0,C 180,E1 -6214.887,E2 -6214.887} C_VEL
LIN {X 0,Y 495.161,Z 469.668,A -85,B 0,C 180,E1 -6216.52,E2 -6216.52} C_VEL
LIN {X 0,Y 495.199,Z 463.964,A -85,B 0,C 180,E1 -6218.159,E2 -6218.159} C_VEL
LIN {X 0,Y 495.317,Z 456.699,A -85,B 0,C 180,E1 -6219.803,E2 -6219.803} C_VEL
LIN {X 0,Y 495.607,Z 448.921,A -85,B 0,C 180,E1 -6221.244,E2 -6221.244} C_VEL
LIN {X 0,Y 495.908,Z 439.538,A -85,B 0,C 180,E1 -6222.689,E2 -6222.689} C_VEL
LIN {X 0,Y 496.348,Z 429.984,A -85,B 0,C 180,E1 -6223.928,E2 -6223.928} C_VEL
LIN {X 0,Y 496.872,Z 417.593,A -85,B 0,C 180,E1 -6225.274,E2 -6225.274} C_VEL
LIN {X 0,Y 497.417,Z 404.943,A -85,B 0,C 180,E1 -6226.414,E2 -6226.414} C_VEL
LIN {X 0,Y 498.047,Z 390.953,A -85,B 0,C 180,E1 -6227.449,E2 -6227.449} C_VEL
LIN {X 0,Y 498.667,Z 377.2,A -85,B 0,C 180,E1 -6228.275,E2 -6228.275} C_VEL
LIN {X 0,Y 499.231,Z 362.741,A -85,B 0,C 180,E1 -6228.966,E2 -6228.966} C_VEL
LIN {X 0,Y 499.693,Z 347.761,A -85,B 0,C 180,E1 -6229.508,E2 -6229.508} C_VEL
LIN {X 0,Y 500.063,Z 332.119,A -85,B 0,C 180,E1 -6229.9,E2 -6229.9} C_VEL
LIN {X 0,Y 501.929,Z 182.93,A -85,B 0,C 180,E1 -6232.282,E2 -6232.282} C_VEL
LIN {X 0,Y 499.207,Z 164.852,A -85,B 0,C 180,E1 -6232.716,E2 -6232.716} C_VEL
LIN {X 0,Y 500.096,Z 142.844,A -85,B 0,C 180,E1 -6234.936,E2 -6234.936} C_VEL
LIN {X 0,Y 500.712,Z 127.665,A -85,B 0,C 180,E1 -6236.485,E2 -6236.485} C_VEL
LIN {X 0,Y 495.76,Z 109.359,A -85,B 0,C 180,E1 -6238.712,E2 -6238.712} C_VEL
LIN {X 0,Y 495.749,Z 109.357,A -85,B 0,C 180,E1 -6241.724,E2 -6241.724} C_VEL
LIN {X 0,Y 495.758,Z 109.357,A -85,B 0,C 180,E1 -6244.692,E2 -6244.692} C_VEL
LIN {X 0,Y 495.72,Z 109.361,A -85,B 0,C 180,E1 -6247.563,E2 -6247.563} C_VEL
LIN {X 0,Y 495.742,Z 109.356,A -85,B 0,C 180,E1 -6250.045,E2 -6250.045} C_VEL
LIN {X 0,Y 495.694,Z 109.367,A -85,B 0,C 180,E1 -6252.887,E2 -6252.887} C_VEL
LIN {X 0,Y 495.721,Z 109.356,A -85,B 0,C 180,E1 -6255.998,E2 -6255.998} C_VEL
LIN {X 0,Y 495.727,Z 109.358,A -85,B 0,C 180,E1 -6259.296,E2 -6259.296} C_VEL
LIN {X 0,Y 495.744,Z 109.357,A -85,B 0,C 180,E1 -6261.408,E2 -6261.408} C_VEL
LIN {X 0,Y 495.742,Z 109.36,A -85,B 0,C 180,E1 -6264.462,E2 -6264.462} C_VEL
LIN {X 0,Y 495.751,Z 109.356,A -85,B 0,C 180,E1 -6267.405,E2 -6267.405} C_VEL
LIN {X 0,Y 495.757,Z 109.36,A -85,B 0,C 180,E1 -6270.253,E2 -6270.253} C_VEL
LIN {X 0,Y 495.739,Z 109.359,A -85,B 0,C 180,E1 -6273.271,E2 -6273.271} C_VEL
LIN {X 0,Y 495.749,Z 109.52,A -85,B 0,C 180,E1 -6276.059,E2 -6276.059} C_VEL
LIN {X 0,Y 497.673,Z 116.802,A -85,B 0,C 180,E1 -6277.202,E2 -6277.202} C_VEL
LIN {X 0,Y 501.505,Z 126.67,A -85,B 0,C 180,E1 -6277.615,E2 -6277.615} C_VEL
LIN {X 0,Y 502.372,Z 130.992,A -85,B 0,C 180,E1 -6277.744,E2 -6277.744} C_VEL
LIN {X 0,Y 500.606,Z 231.28,A -85,B 0,C 180,E1 -6279.48,E2 -6279.48} C_VEL
LIN {X 0,Y 500.007,Z 281.594,A -85,B 0,C 180,E1 -6280.32,E2 -6280.32} C_VEL
LIN {X 0,Y 499.722,Z 296.528,A -85,B 0,C 180,E1 -6280.719,E2 -6280.719} C_VEL
LIN {X 0,Y 499.331,Z 311.207,A -85,B 0,C 180,E1 -6281.272,E2 -6281.272} C_VEL
LIN {X 0,Y 498.925,Z 324.955,A -85,B 0,C 180,E1 -6281.947,E2 -6281.947} C_VEL
LIN {X 0,Y 498.384,Z 338.475,A -85,B 0,C 180,E1 -6282.775,E2 -6282.775} C_VEL
LIN {X 0,Y 497.838,Z 351.245,A -85,B 0,C 180,E1 -6283.732,E2 -6283.732} C_VEL
LIN {X 0,Y 497.295,Z 363.535,A -85,B 0,C 180,E1 -6284.844,E2 -6284.844} C_VEL
LIN {X 0,Y 496.8,Z 374.948,A -85,B 0,C 180,E1 -6286.085,E2 -6286.085} C_VEL
LIN {X 0,Y 496.402,Z 384.518,A -85,B 0,C 180,E1 -6287.324,E2 -6287.324} C_VEL
LIN {X 0,Y 496.015,Z 393.859,A -85,B 0,C 180,E1 -6288.766,E2 -6288.766} C_VEL
LIN {X 0,Y 495.639,Z 401.595,A -85,B 0,C 180,E1 -6290.203,E2 -6290.203} C_VEL
LIN {X 0,Y 495.425,Z 408.763,A -85,B 0,C 180,E1 -6291.845,E2 -6291.845} C_VEL
LIN {X 0,Y 495.251,Z 414.383,A -85,B 0,C 180,E1 -6293.482,E2 -6293.482} C_VEL
LIN {X 0,Y 495.05,Z 418.618,A -85,B 0,C 180,E1 -6295.114,E2 -6295.114} C_VEL
LIN {X 0,Y 495.143,Z 421.569,A -85,B 0,C 180,E1 -6296.746,E2 -6296.746} C_VEL
LIN {X 0,Y 494.964,Z 423.341,A -85,B 0,C 180,E1 -6298.373,E2 -6298.373} C_VEL
LIN {X 0,Y 494.916,Z 423.925,A -85,B 0,C 180,E1 -6300,E2 -6300} C_VEL
LIN {X 0,Y 494.964,Z 423.318,A -85,B 0,C 180,E1 -6301.628,E2 -6301.628} C_VEL
LIN {X 0,Y 495.132,Z 421.55,A -85,B 0,C 180,E1 -6303.255,E2 -6303.255} C_VEL
LIN {X 0,Y 495.039,Z 418.604,A -85,B 0,C 180,E1 -6304.887,E2 -6304.887} C_VEL
LIN {X 0,Y 495.218,Z 415.031,A -85,B 0,C 180,E1 -6306.304,E2 -6306.304} C_VEL
LIN {X 0,Y 495.328,Z 410.352,A -85,B 0,C 180,E1 -6307.747,E2 -6307.747} C_VEL
LIN {X 0,Y 495.54,Z 403.649,A -85,B 0,C 180,E1 -6309.387,E2 -6309.387} C_VEL
LIN {X 0,Y 495.848,Z 396.382,A -85,B 0,C 180,E1 -6310.825,E2 -6310.825} C_VEL
LIN {X 0,Y 496.129,Z 387.634,A -85,B 0,C 180,E1 -6312.268,E2 -6312.268} C_VEL
LIN {X 0,Y 496.582,Z 378.701,A -85,B 0,C 180,E1 -6313.505,E2 -6313.505} C_VEL
LIN {X 0,Y 497.076,Z 368.144,A -85,B 0,C 180,E1 -6314.744,E2 -6314.744} C_VEL
LIN {X 0,Y 497.652,Z 355.826,A -85,B 0,C 180,E1 -6315.953,E2 -6315.953} C_VEL
LIN {X 0,Y 498.236,Z 342.701,A -85,B 0,C 180,E1 -6317.02,E2 -6317.02} C_VEL
LIN {X 0,Y 498.746,Z 330.357,A -85,B 0,C 180,E1 -6317.848,E2 -6317.848} C_VEL
LIN {X 0,Y 499.256,Z 316.08,A -85,B 0,C 180,E1 -6318.625,E2 -6318.625} C_VEL
LIN {X 0,Y 499.74,Z 300.527,A -85,B 0,C 180,E1 -6319.277,E2 -6319.277} C_VEL
LIN {X 0,Y 500.1,Z 285.318,A -85,B 0,C 180,E1 -6319.738,E2 -6319.738} C_VEL
LIN {X 0,Y 500.293,Z 269.559,A -85,B 0,C 180,E1 -6320.051,E2 -6320.051} C_VEL
LIN {X 0,Y 502.04,Z 130.405,A -85,B 0,C 180,E1 -6322.262,E2 -6322.262} C_VEL
LIN {X 0,Y 500.217,Z 123.189,A -85,B 0,C 180,E1 -6322.47,E2 -6322.47} C_VEL
LIN {X 0,Y 496.73,Z 113.898,A -85,B 0,C 180,E1 -6322.808,E2 -6322.808} C_VEL
LIN {X 0,Y 495.75,Z 109.36,A -85,B 0,C 180,E1 -6323.581,E2 -6323.581} C_VEL
LIN {X 0,Y 495.748,Z 109.355,A -85,B 0,C 180,E1 -6326.978,E2 -6326.978} C_VEL
LIN {X 0,Y 495.761,Z 109.356,A -85,B 0,C 180,E1 -6330.146,E2 -6330.146} C_VEL
LIN {X 0,Y 495.753,Z 109.357,A -85,B 0,C 180,E1 -6333.237,E2 -6333.237} C_VEL
LIN {X 0,Y 495.713,Z 109.36,A -85,B 0,C 180,E1 -6336.087,E2 -6336.087} C_VEL
LIN {X 0,Y 495.76,Z 109.353,A -85,B 0,C 180,E1 -6338.767,E2 -6338.767} C_VEL
LIN {X 0,Y 495.738,Z 109.358,A -85,B 0,C 180,E1 -6339.417,E2 -6339.417} C_VEL
LIN {X 0,Y 495.084,Z 109.445,A -85,B 0,C 180,E1 -6340.095,E2 -6340.095} C_VEL
LIN {X 0,Y 492.223,Z 109.802,A -85,B 0,C 180,E1 -6341.196,E2 -6341.196} C_VEL
LIN {X 0,Y 489.794,Z 110.101,A -85,B 0,C 180,E1 -6342.083,E2 -6342.083} C_VEL
LIN {X 0,Y 488.746,Z 110.227,A -85,B 0,C 180,E1 -6342.768,E2 -6342.768} C_VEL
LIN {X 0,Y 488.659,Z 110.237,A -85,B 0,C 180,E1 -6343,E2 -6343} C_VEL
LIN {X 0,Y 488.69,Z 110.221,A -85,B 0,C 180,E1 -6345.978,E2 -6345.978} C_VEL
LIN {X 0,Y 488.664,Z 110.232,A -85,B 0,C 180,E1 -6348.58,E2 -6348.58} C_VEL
LIN {X 0,Y 488.7,Z 110.237,A -85,B 0,C 180,E1 -6350.949,E2 -6350.949} C_VEL
LIN {X 0,Y 488.671,Z 110.226,A -85,B 0,C 180,E1 -6353.867,E2 -6353.867} C_VEL
LIN {X 0,Y 488.704,Z 110.235,A -85,B 0,C 180,E1 -6356.875,E2 -6356.875} C_VEL
LIN {X 0,Y 488.706,Z 110.226,A -85,B 0,C 180,E1 -6359.779,E2 -6359.779} C_VEL
LIN {X 0,Y 488.701,Z 110.237,A -85,B 0,C 180,E1 -6363.079,E2 -6363.079} C_VEL
LIN {X 0,Y 488.698,Z 110.227,A -85,B 0,C 180,E1 -6365.351,E2 -6365.351} C_VEL
LIN {X 0,Y 488.69,Z 110.234,A -85,B 0,C 180,E1 -6368.043,E2 -6368.043} C_VEL
LIN {X 0,Y 488.73,Z 110.231,A -85,B 0,C 180,E1 -6370.686,E2 -6370.686} C_VEL
LIN {X 0,Y 488.679,Z 110.232,A -85,B 0,C 180,E1 -6373.284,E2 -6373.284} C_VEL
LIN {X 0,Y 488.715,Z 110.232,A -85,B 0,C 180,E1 -6375.849,E2 -6375.849} C_VEL
LIN {X 0,Y 488.809,Z 110.226,A -85,B 0,C 180,E1 -6378.388,E2 -6378.388} C_VEL
LIN {X 0,Y 488.761,Z 110.226,A -85,B 0,C 180,E1 -6381.733,E2 -6381.733} C_VEL
LIN {X 0,Y 488.807,Z 110.225,A -85,B 0,C 180,E1 -6384.224,E2 -6384.224} C_VEL
LIN {X 0,Y 488.943,Z 110.207,A -85,B 0,C 180,E1 -6387.529,E2 -6387.529} C_VEL
LIN {X 0,Y 488.803,Z 110.418,A -85,B 0,C 180,E1 -6389.485,E2 -6389.485} C_VEL
LIN {X 0,Y 491.985,Z 124.548,A -85,B 0,C 180,E1 -6391.637,E2 -6391.637} C_VEL
LIN {X 0,Y 492.048,Z 130.401,A -85,B 0,C 180,E1 -6392.456,E2 -6392.456} C_VEL
LIN {X 0,Y 491.764,Z 141.749,A -85,B 0,C 180,E1 -6394.021,E2 -6394.021} C_VEL
LIN {X 0,Y 495.552,Z 159.488,A -85,B 0,C 180,E1 -6394.489,E2 -6394.489} C_VEL
LIN {X 0,Y 494.075,Z 307.434,A -85,B 0,C 180,E1 -6396.714,E2 -6396.714} C_VEL
LIN {X 0,Y 493.737,Z 322.783,A -85,B 0,C 180,E1 -6397.103,E2 -6397.103} C_VEL
LIN {X 0,Y 493.307,Z 337.06,A -85,B 0,C 180,E1 -6397.624,E2 -6397.624} C_VEL
LIN {X 0,Y 492.718,Z 351.227,A -85,B 0,C 180,E1 -6398.304,E2 -6398.304} C_VEL
LIN {X 0,Y 492.055,Z 364.868,A -85,B 0,C 180,E1 -6399.131,E2 -6399.131} C_VEL
LIN {X 0,Y 491.443,Z 377.679,A -85,B 0,C 180,E1 -6400.089,E2 -6400.089} C_VEL
LIN {X 0,Y 490.718,Z 389.499,A -85,B 0,C 180,E1 -6401.148,E2 -6401.148} C_VEL
LIN {X 0,Y 490.089,Z 401.315,A -85,B 0,C 180,E1 -6402.422,E2 -6402.422} C_VEL
LIN {X 0,Y 489.523,Z 411.302,A -85,B 0,C 180,E1 -6403.703,E2 -6403.703} C_VEL
LIN {X 0,Y 488.946,Z 421.587,A -85,B 0,C 180,E1 -6405.294,E2 -6405.294} C_VEL
LIN {X 0,Y 488.55,Z 430.258,A -85,B 0,C 180,E1 -6406.936,E2 -6406.936} C_VEL
LIN {X 0,Y 488.315,Z 436.828,A -85,B 0,C 180,E1 -6408.459,E2 -6408.459} C_VEL
LIN {X 0,Y 488.096,Z 442.834,A -85,B 0,C 180,E1 -6410.217,E2 -6410.217} C_VEL
LIN {X 0,Y 487.947,Z 447.383,A -85,B 0,C 180,E1 -6411.992,E2 -6411.992} C_VEL
LIN {X 0,Y 487.797,Z 450.545,A -85,B 0,C 180,E1 -6413.792,E2 -6413.792} C_VEL
LIN {X 0,Y 487.775,Z 452.325,A -85,B 0,C 180,E1 -6415.61,E2 -6415.61} C_VEL
LIN {X 0,Y 487.776,Z 452.721,A -85,B 0,C 180,E1 -6417.456,E2 -6417.456} C_VEL
LIN {X 0,Y 487.825,Z 452.32,A -85,B 0,C 180,E1 -6418.499,E2 -6418.499} C_VEL
LIN {X 0,Y 487.872,Z 450.587,A -85,B 0,C 180,E1 -6420.278,E2 -6420.278} C_VEL
LIN {X 0,Y 487.962,Z 447.201,A -85,B 0,C 180,E1 -6422.202,E2 -6422.202} C_VEL
LIN {X 0,Y 488.064,Z 443.313,A -85,B 0,C 180,E1 -6423.726,E2 -6423.726} C_VEL
LIN {X 0,Y 488.235,Z 438.67,A -85,B 0,C 180,E1 -6425.155,E2 -6425.155} C_VEL
LIN {X 0,Y 488.456,Z 432.432,A -85,B 0,C 180,E1 -6426.703,E2 -6426.703} C_VEL
LIN {X 0,Y 488.81,Z 425.114,A -85,B 0,C 180,E1 -6428.188,E2 -6428.188} C_VEL
LIN {X 0,Y 489.208,Z 415.854,A -85,B 0,C 180,E1 -6429.739,E2 -6429.739} C_VEL
LIN {X 0,Y 489.81,Z 406.356,A -85,B 0,C 180,E1 -6431.064,E2 -6431.064} C_VEL
LIN {X 0,Y 490.418,Z 395.483,A -85,B 0,C 180,E1 -6432.341,E2 -6432.341} C_VEL
LIN {X 0,Y 491.072,Z 383.359,A -85,B 0,C 180,E1 -6433.531,E2 -6433.531} C_VEL
LIN {X 0,Y 491.805,Z 370.283,A -85,B 0,C 180,E1 -6434.588,E2 -6434.588} C_VEL
LIN {X 0,Y 492.447,Z 357.266,A -85,B 0,C 180,E1 -6435.454,E2 -6435.454} C_VEL
LIN {X 0,Y 493.054,Z 343.278,A -85,B 0,C 180,E1 -6436.201,E2 -6436.201} C_VEL
LIN {X 0,Y 493.587,Z 328.039,A -85,B 0,C 180,E1 -6436.823,E2 -6436.823} C_VEL
LIN {X 0,Y 493.992,Z 313.152,A -85,B 0,C 180,E1 -6437.258,E2 -6437.258} C_VEL
LIN {X 0,Y 494.248,Z 295.334,A -85,B 0,C 180,E1 -6437.58,E2 -6437.58} C_VEL
LIN {X 0,Y 495.523,Z 155.609,A -85,B 0,C 180,E1 -6439.676,E2 -6439.676} C_VEL
LIN {X 0,Y 492.817,Z 140.123,A -85,B 0,C 180,E1 -6440.078,E2 -6440.078} C_VEL
LIN {X 0,Y 493.09,Z 127.502,A -85,B 0,C 180,E1 -6441.44,E2 -6441.44} C_VEL
LIN {X 0,Y 489.156,Z 111.953,A -85,B 0,C 180,E1 -6443.32,E2 -6443.32} C_VEL
LIN {X 0,Y 488.706,Z 110.237,A -85,B 0,C 180,E1 -6443.535,E2 -6443.535} C_VEL
LIN {X 0,Y 488.737,Z 110.231,A -85,B 0,C 180,E1 -6446.516,E2 -6446.516} C_VEL
LIN {X 0,Y 488.727,Z 110.234,A -85,B 0,C 180,E1 -6449.781,E2 -6449.781} C_VEL
LIN {X 0,Y 488.795,Z 110.225,A -85,B 0,C 180,E1 -6453.056,E2 -6453.056} C_VEL
LIN {X 0,Y 488.7,Z 110.237,A -85,B 0,C 180,E1 -6456.255,E2 -6456.255} C_VEL
LIN {X 0,Y 488.743,Z 110.446,A -85,B 0,C 180,E1 -6456.484,E2 -6456.484} C_VEL
LIN {X 0,Y 489.5,Z 113.574,A -85,B 0,C 180,E1 -6456.928,E2 -6456.928} C_VEL
LIN {X 0,Y 495.522,Z 128.948,A -85,B 0,C 180,E1 -6457.484,E2 -6457.484} C_VEL
LIN {X 0,Y 493.451,Z 280.971,A -85,B 0,C 180,E1 -6459.985,E2 -6459.985} C_VEL
LIN {X 0,Y 493.108,Z 296.618,A -85,B 0,C 180,E1 -6460.415,E2 -6460.415} C_VEL
LIN {X 0,Y 492.644,Z 311.814,A -85,B 0,C 180,E1 -6461.007,E2 -6461.007} C_VEL
LIN {X 0,Y 492.163,Z 325.305,A -85,B 0,C 180,E1 -6461.69,E2 -6461.69} C_VEL
LIN {X 0,Y 491.573,Z 338.643,A -85,B 0,C 180,E1 -6462.528,E2 -6462.528} C_VEL
LIN {X 0,Y 490.966,Z 351.942,A -85,B 0,C 180,E1 -6463.553,E2 -6463.553} C_VEL
LIN {X 0,Y 490.403,Z 364.53,A -85,B 0,C 180,E1 -6464.732,E2 -6464.732} C_VEL
LIN {X 0,Y 489.855,Z 374.883,A -85,B 0,C 180,E1 -6465.883,E2 -6465.883} C_VEL
LIN {X 0,Y 489.293,Z 385.926,A -85,B 0,C 180,E1 -6467.347,E2 -6467.347} C_VEL
LIN {X 0,Y 488.951,Z 395.049,A -85,B 0,C 180,E1 -6468.811,E2 -6468.811} C_VEL
LIN {X 0,Y 488.588,Z 401.581,A -85,B 0,C 180,E1 -6470.06,E2 -6470.06} C_VEL
LIN {X 0,Y 488.353,Z 408.821,A -85,B 0,C 180,E1 -6471.725,E2 -6471.725} C_VEL
LIN {X 0,Y 488.145,Z 414.632,A -85,B 0,C 180,E1 -6473.423,E2 -6473.423} C_VEL
LIN {X 0,Y 487.976,Z 418.833,A -85,B 0,C 180,E1 -6475.042,E2 -6475.042} C_VEL
LIN {X 0,Y 488.06,Z 421.869,A -85,B 0,C 180,E1 -6476.698,E2 -6476.698} C_VEL
LIN {X 0,Y 487.893,Z 423.728,A -85,B 0,C 180,E1 -6478.349,E2 -6478.349} C_VEL
LIN {X 0,Y 487.838,Z 424.408,A -85,B 0,C 180,E1 -6480,E2 -6480} C_VEL
LIN {X 0,Y 487.895,Z 423.879,A -85,B 0,C 180,E1 -6481.651,E2 -6481.651} C_VEL
LIN {X 0,Y 488.074,Z 422.181,A -85,B 0,C 180,E1 -6483.302,E2 -6483.302} C_VEL
LIN {X 0,Y 487.995,Z 419.298,A -85,B 0,C 180,E1 -6484.957,E2 -6484.957} C_VEL
LIN {X 0,Y 488.22,Z 415.126,A -85,B 0,C 180,E1 -6486.613,E2 -6486.613} C_VEL
LIN {X 0,Y 488.403,Z 409.579,A -85,B 0,C 180,E1 -6488.273,E2 -6488.273} C_VEL
LIN {X 0,Y 488.621,Z 402.496,A -85,B 0,C 180,E1 -6489.939,E2 -6489.939} C_VEL
LIN {X 0,Y 488.989,Z 394.85,A -85,B 0,C 180,E1 -6491.398,E2 -6491.398} C_VEL
LIN {X 0,Y 489.348,Z 385.593,A -85,B 0,C 180,E1 -6492.862,E2 -6492.862} C_VEL
LIN {X 0,Y 489.864,Z 376.152,A -85,B 0,C 180,E1 -6494.116,E2 -6494.116} C_VEL
LIN {X 0,Y 490.412,Z 364.872,A -85,B 0,C 180,E1 -6495.374,E2 -6495.374} C_VEL
LIN {X 0,Y 491.033,Z 353.047,A -85,B 0,C 180,E1 -6496.473,E2 -6496.473} C_VEL
LIN {X 0,Y 491.549,Z 340.197,A -85,B 0,C 180,E1 -6497.472,E2 -6497.472} C_VEL
LIN {X 0,Y 492.132,Z 326.955,A -85,B 0,C 180,E1 -6498.311,E2 -6498.311} C_VEL
LIN {X 0,Y 492.564,Z 313.562,A -85,B 0,C 180,E1 -6498.995,E2 -6498.995} C_VEL
LIN {X 0,Y 493.001,Z 298.82,A -85,B 0,C 180,E1 -6499.579,E2 -6499.579} C_VEL
LIN {X 0,Y 493.287,Z 283.25,A -85,B 0,C 180,E1 -6500.022,E2 -6500.022} C_VEL
LIN {X 0,Y 495.476,Z 158.856,A -85,B 0,C 180,E1 -6502.208,E2 -6502.208} C_VEL
LIN {X 0,Y 495.991,Z 131.521,A -85,B 0,C 180,E1 -6502.721,E2 -6502.721} C_VEL
LIN {X 0,Y 494.03,Z 126.267,A -85,B 0,C 180,E1 -6502.944,E2 -6502.944} C_VEL
LIN {X 0,Y 490.9,Z 119.122,A -85,B 0,C 180,E1 -6503.293,E2 -6503.293} C_VEL
LIN {X 0,Y 488.68,Z 110.242,A -85,B 0,C 180,E1 -6505.255,E2 -6505.255} C_VEL
LIN {X 0,Y 488.698,Z 110.239,A -85,B 0,C 180,E1 -6507.399,E2 -6507.399} C_VEL
LIN {X 0,Y 488.704,Z 110.235,A -85,B 0,C 180,E1 -6510.361,E2 -6510.361} C_VEL
LIN {X 0,Y 488.709,Z 110.237,A -85,B 0,C 180,E1 -6513.479,E2 -6513.479} C_VEL
LIN {X 0,Y 488.672,Z 110.238,A -85,B 0,C 180,E1 -6516.353,E2 -6516.353} C_VEL
LIN {X 0,Y 488.694,Z 110.239,A -85,B 0,C 180,E1 -6519.255,E2 -6519.255} C_VEL
LIN {X 0,Y 488.649,Z 110.241,A -85,B 0,C 180,E1 -6522.53,E2 -6522.53} C_VEL
LIN {X 0,Y 488.7,Z 110.238,A -85,B 0,C 180,E1 -6525.197,E2 -6525.197} C_VEL
LIN {X 0,Y 488.661,Z 110.24,A -85,B 0,C 180,E1 -6528.579,E2 -6528.579} C_VEL
LIN {X 0,Y 488.697,Z 110.239,A -85,B 0,C 180,E1 -6530.948,E2 -6530.948} C_VEL
LIN {X 0,Y 488.664,Z 110.241,A -85,B 0,C 180,E1 -6533.867,E2 -6533.867} C_VEL
LIN {X 0,Y 488.7,Z 110.239,A -85,B 0,C 180,E1 -6536.874,E2 -6536.874} C_VEL
LIN {X 0,Y 488.697,Z 110.279,A -85,B 0,C 180,E1 -6538.978,E2 -6538.978} C_VEL
LIN {X 0,Y 491.988,Z 122.962,A -85,B 0,C 180,E1 -6541.176,E2 -6541.176} C_VEL
LIN {X 0,Y 493.094,Z 128.721,A -85,B 0,C 180,E1 -6542.089,E2 -6542.089} C_VEL
LIN {X 0,Y 492.125,Z 147.14,A -85,B 0,C 180,E1 -6544.632,E2 -6544.632} C_VEL
LIN {X 0,Y 491.411,Z 163.154,A -85,B 0,C 180,E1 -6546.751,E2 -6546.751} C_VEL
LIN {X 0,Y 495.007,Z 184.542,A -85,B 0,C 180,E1 -6547.377,E2 -6547.377} C_VEL
LIN {X 0,Y 495.398,Z 188.735,A -85,B 0,C 180,E1 -6547.478,E2 -6547.478} C_VEL
LIN {X 0,Y 493.683,Z 288.764,A -85,B 0,C 180,E1 -6549.233,E2 -6549.233} C_VEL
LIN {X 0,Y 493.011,Z 333.24,A -85,B 0,C 180,E1 -6549.993,E2 -6549.993} C_VEL
LIN {X 0,Y 492.522,Z 349.162,A -85,B 0,C 180,E1 -6550.435,E2 -6550.435} C_VEL
LIN {X 0,Y 492.013,Z 364.538,A -85,B 0,C 180,E1 -6551.037,E2 -6551.037} C_VEL
LIN {X 0,Y 491.425,Z 379.315,A -85,B 0,C 180,E1 -6551.77,E2 -6551.77} C_VEL
LIN {X 0,Y 490.845,Z 392.877,A -85,B 0,C 180,E1 -6552.609,E2 -6552.609} C_VEL
LIN {X 0,Y 490.282,Z 406.374,A -85,B 0,C 180,E1 -6553.64,E2 -6553.64} C_VEL
LIN {X 0,Y 489.698,Z 418.996,A -85,B 0,C 180,E1 -6554.816,E2 -6554.816} C_VEL
LIN {X 0,Y 489.234,Z 430.22,A -85,B 0,C 180,E1 -6556.077,E2 -6556.077} C_VEL
LIN {X 0,Y 488.787,Z 441.086,A -85,B 0,C 180,E1 -6557.545,E2 -6557.545} C_VEL
LIN {X 0,Y 488.44,Z 450.079,A -85,B 0,C 180,E1 -6559.009,E2 -6559.009} C_VEL
LIN {X 0,Y 488.185,Z 457.583,A -85,B 0,C 180,E1 -6560.47,E2 -6560.47} C_VEL
LIN {X 0,Y 488.066,Z 464.627,A -85,B 0,C 180,E1 -6562.137,E2 -6562.137} C_VEL
LIN {X 0,Y 488.013,Z 469.41,A -85,B 0,C 180,E1 -6563.558,E2 -6563.558} C_VEL
LIN {X 0,Y 487.941,Z 473.29,A -85,B 0,C 180,E1 -6565.042,E2 -6565.042} C_VEL
LIN {X 0,Y 487.955,Z 476.405,A -85,B 0,C 180,E1 -6566.697,E2 -6566.697} C_VEL
LIN {X 0,Y 487.89,Z 478.271,A -85,B 0,C 180,E1 -6568.349,E2 -6568.349} C_VEL
LIN {X 0,Y 487.828,Z 478.933,A -85,B 0,C 180,E1 -6570,E2 -6570} C_VEL
LIN {X 0,Y 487.89,Z 478.352,A -85,B 0,C 180,E1 -6571.651,E2 -6571.651} C_VEL
LIN {X 0,Y 487.954,Z 476.567,A -85,B 0,C 180,E1 -6573.303,E2 -6573.303} C_VEL
LIN {X 0,Y 487.933,Z 473.549,A -85,B 0,C 180,E1 -6574.958,E2 -6574.958} C_VEL
LIN {X 0,Y 488.069,Z 469.241,A -85,B 0,C 180,E1 -6576.615,E2 -6576.615} C_VEL
LIN {X 0,Y 488.102,Z 463.512,A -85,B 0,C 180,E1 -6578.279,E2 -6578.279} C_VEL
LIN {X 0,Y 488.263,Z 456.22,A -85,B 0,C 180,E1 -6579.946,E2 -6579.946} C_VEL
LIN {X 0,Y 488.573,Z 448.409,A -85,B 0,C 180,E1 -6581.408,E2 -6581.408} C_VEL
LIN {X 0,Y 488.876,Z 438.981,A -85,B 0,C 180,E1 -6582.875,E2 -6582.875} C_VEL
LIN {X 0,Y 489.34,Z 429.387,A -85,B 0,C 180,E1 -6584.132,E2 -6584.132} C_VEL
LIN {X 0,Y 489.874,Z 417.982,A -85,B 0,C 180,E1 -6585.391,E2 -6585.391} C_VEL
LIN {X 0,Y 490.449,Z 405.305,A -85,B 0,C 180,E1 -6586.561,E2 -6586.561} C_VEL
LIN {X 0,Y 491.103,Z 391.676,A -85,B 0,C 180,E1 -6587.597,E2 -6587.597} C_VEL
LIN {X 0,Y 491.768,Z 378.176,A -85,B 0,C 180,E1 -6588.433,E2 -6588.433} C_VEL
LIN {X 0,Y 492.378,Z 363.342,A -85,B 0,C 180,E1 -6589.165,E2 -6589.165} C_VEL
LIN {X 0,Y 492.901,Z 347.995,A -85,B 0,C 180,E1 -6589.737,E2 -6589.737} C_VEL
LIN {X 0,Y 493.306,Z 332.927,A -85,B 0,C 180,E1 -6590.13,E2 -6590.13} C_VEL
LIN {X 0,Y 495.316,Z 183.828,A -85,B 0,C 180,E1 -6592.567,E2 -6592.567} C_VEL
LIN {X 0,Y 492.448,Z 164.38,A -85,B 0,C 180,E1 -6593.058,E2 -6593.058} C_VEL
LIN {X 0,Y 493.4,Z 142.455,A -85,B 0,C 180,E1 -6595.298,E2 -6595.298} C_VEL
LIN {X 0,Y 493.972,Z 129.579,A -85,B 0,C 180,E1 -6596.626,E2 -6596.626} C_VEL
LIN {X 0,Y 488.723,Z 110.235,A -85,B 0,C 180,E1 -6599.006,E2 -6599.006} C_VEL
LIN {X 0,Y 488.694,Z 110.235,A -85,B 0,C 180,E1 -6602.148,E2 -6602.148} C_VEL
LIN {X 0,Y 488.711,Z 110.236,A -85,B 0,C 180,E1 -6605.116,E2 -6605.116} C_VEL
LIN {X 0,Y 488.673,Z 110.238,A -85,B 0,C 180,E1 -6608.201,E2 -6608.201} C_VEL
LIN {X 0,Y 488.692,Z 110.236,A -85,B 0,C 180,E1 -6610.341,E2 -6610.341} C_VEL
LIN {X 0,Y 488.672,Z 110.235,A -85,B 0,C 180,E1 -6613.656,E2 -6613.656} C_VEL
LIN {X 0,Y 488.672,Z 110.237,A -85,B 0,C 180,E1 -6616.344,E2 -6616.344} C_VEL
LIN {X 0,Y 488.703,Z 110.233,A -85,B 0,C 180,E1 -6619.674,E2 -6619.674} C_VEL
LIN {X 0,Y 488.669,Z 110.241,A -85,B 0,C 180,E1 -6622.84,E2 -6622.84} C_VEL
LIN {X 0,Y 488.717,Z 110.232,A -85,B 0,C 180,E1 -6625.886,E2 -6625.886} C_VEL
LIN {X 0,Y 488.689,Z 110.239,A -85,B 0,C 180,E1 -6628.82,E2 -6628.82} C_VEL
LIN {X 0,Y 488.695,Z 110.237,A -85,B 0,C 180,E1 -6631.668,E2 -6631.668} C_VEL
LIN {X 0,Y 488.698,Z 110.238,A -85,B 0,C 180,E1 -6634.959,E2 -6634.959} C_VEL
LIN {X 0,Y 488.72,Z 110.423,A -85,B 0,C 180,E1 -6635.692,E2 -6635.692} C_VEL
LIN {X 0,Y 490.592,Z 117.369,A -85,B 0,C 180,E1 -6636.795,E2 -6636.795} C_VEL
LIN {X 0,Y 495.303,Z 128.841,A -85,B 0,C 180,E1 -6637.309,E2 -6637.309} C_VEL
LIN {X 0,Y 495.943,Z 131.674,A -85,B 0,C 180,E1 -6637.403,E2 -6637.403} C_VEL
LIN {X 0,Y 494.025,Z 230.099,A -85,B 0,C 180,E1 -6639.167,E2 -6639.167} C_VEL
LIN {X 0,Y 493.296,Z 282.518,A -85,B 0,C 180,E1 -6640.069,E2 -6640.069} C_VEL
LIN {X 0,Y 492.95,Z 297.953,A -85,B 0,C 180,E1 -6640.496,E2 -6640.496} C_VEL
LIN {X 0,Y 492.539,Z 313.618,A -85,B 0,C 180,E1 -6641.112,E2 -6641.112} C_VEL
LIN {X 0,Y 492.094,Z 326.9,A -85,B 0,C 180,E1 -6641.795,E2 -6641.795} C_VEL
LIN {X 0,Y 491.54,Z 340.106,A -85,B 0,C 180,E1 -6642.635,E2 -6642.635} C_VEL
LIN {X 0,Y 490.881,Z 353.763,A -85,B 0,C 180,E1 -6643.695,E2 -6643.695} C_VEL
LIN {X 0,Y 490.305,Z 365.833,A -85,B 0,C 180,E1 -6644.836,E2 -6644.836} C_VEL
LIN {X 0,Y 489.808,Z 376.934,A -85,B 0,C 180,E1 -6646.094,E2 -6646.094} C_VEL
LIN {X 0,Y 489.292,Z 387.689,A -85,B 0,C 180,E1 -6647.558,E2 -6647.558} C_VEL
LIN {X 0,Y 488.896,Z 396.57,A -85,B 0,C 180,E1 -6649.02,E2 -6649.02} C_VEL
LIN {X 0,Y 488.555,Z 403.904,A -85,B 0,C 180,E1 -6650.478,E2 -6650.478} C_VEL
LIN {X 0,Y 488.335,Z 410.691,A -85,B 0,C 180,E1 -6652.142,E2 -6652.142} C_VEL
LIN {X 0,Y 488.196,Z 415.501,A -85,B 0,C 180,E1 -6653.644,E2 -6653.644} C_VEL
LIN {X 0,Y 487.981,Z 418.997,A -85,B 0,C 180,E1 -6655.043,E2 -6655.043} C_VEL
LIN {X 0,Y 488.06,Z 421.957,A -85,B 0,C 180,E1 -6656.698,E2 -6656.698} C_VEL
LIN {X 0,Y 487.894,Z 423.73,A -85,B 0,C 180,E1 -6658.349,E2 -6658.349} C_VEL
LIN {X 0,Y 487.836,Z 424.31,A -85,B 0,C 180,E1 -6660,E2 -6660} C_VEL
LIN {X 0,Y 487.894,Z 423.692,A -85,B 0,C 180,E1 -6661.651,E2 -6661.651} C_VEL
LIN {X 0,Y 488.05,Z 421.908,A -85,B 0,C 180,E1 -6663.302,E2 -6663.302} C_VEL
LIN {X 0,Y 487.97,Z 418.936,A -85,B 0,C 180,E1 -6664.958,E2 -6664.958} C_VEL
LIN {X 0,Y 488.148,Z 414.788,A -85,B 0,C 180,E1 -6666.58,E2 -6666.58} C_VEL
LIN {X 0,Y 488.33,Z 409.066,A -85,B 0,C 180,E1 -6668.275,E2 -6668.275} C_VEL
LIN {X 0,Y 488.575,Z 401.913,A -85,B 0,C 180,E1 -6669.94,E2 -6669.94} C_VEL
LIN {X 0,Y 488.926,Z 394.216,A -85,B 0,C 180,E1 -6671.4,E2 -6671.4} C_VEL
LIN {X 0,Y 489.281,Z 386.403,A -85,B 0,C 180,E1 -6672.654,E2 -6672.654} C_VEL
LIN {X 0,Y 489.779,Z 375.463,A -85,B 0,C 180,E1 -6674.119,E2 -6674.119} C_VEL
LIN {X 0,Y 490.34,Z 364.197,A -85,B 0,C 180,E1 -6675.377,E2 -6675.377} C_VEL
LIN {X 0,Y 490.953,Z 351.861,A -85,B 0,C 180,E1 -6676.526,E2 -6676.526} C_VEL
LIN {X 0,Y 491.536,Z 339.685,A -85,B 0,C 180,E1 -6677.473,E2 -6677.473} C_VEL
LIN {X 0,Y 492.074,Z 326.639,A -85,B 0,C 180,E1 -6678.314,E2 -6678.314} C_VEL
LIN {X 0,Y 492.643,Z 312.382,A -85,B 0,C 180,E1 -6679.047,E2 -6679.047} C_VEL
LIN {X 0,Y 493.082,Z 296.719,A -85,B 0,C 180,E1 -6679.661,E2 -6679.661} C_VEL
LIN {X 0,Y 493.399,Z 282.087,A -85,B 0,C 180,E1 -6680.072,E2 -6680.072} C_VEL
LIN {X 0,Y 493.668,Z 259.372,A -85,B 0,C 180,E1 -6680.468,E2 -6680.468} C_VEL
LIN {X 0,Y 495.434,Z 131.918,A -85,B 0,C 180,E1 -6682.543,E2 -6682.543} C_VEL
LIN {X 0,Y 493.975,Z 125.819,A -85,B 0,C 180,E1 -6682.714,E2 -6682.714} C_VEL
LIN {X 0,Y 489.625,Z 114.235,A -85,B 0,C 180,E1 -6683.131,E2 -6683.131} C_VEL
LIN {X 0,Y 488.728,Z 110.236,A -85,B 0,C 180,E1 -6683.8,E2 -6683.8} C_VEL
LIN {X 0,Y 488.714,Z 110.232,A -85,B 0,C 180,E1 -6686.925,E2 -6686.925} C_VEL
LIN {X 0,Y 488.72,Z 110.232,A -85,B 0,C 180,E1 -6690.22,E2 -6690.22} C_VEL
LIN {X 0,Y 488.712,Z 110.237,A -85,B 0,C 180,E1 -6693.48,E2 -6693.48} C_VEL
LIN {X 0,Y 488.675,Z 110.235,A -85,B 0,C 180,E1 -6696.353,E2 -6696.353} C_VEL
LIN {X 0,Y 488.686,Z 110.236,A -85,B 0,C 180,E1 -6699.413,E2 -6699.413} C_VEL
LIN {X 0,Y 488.666,Z 110.237,A -85,B 0,C 180,E1 -6702.821,E2 -6702.821} C_VEL
LIN {X 0,Y 488.659,Z 110.237,A -85,B 0,C 180,E1 -6703,E2 -6703} C_VEL
LIN {X 0,Y 487.984,Z 110.322,A -85,B 0,C 180,E1 -6703.688,E2 -6703.688} C_VEL
LIN {X 0,Y 485.117,Z 110.677,A -85,B 0,C 180,E1 -6704.805,E2 -6704.805} C_VEL
LIN {X 0,Y 482.708,Z 110.969,A -85,B 0,C 180,E1 -6705.705,E2 -6705.705} C_VEL
LIN {X 0,Y 481.691,Z 111.092,A -85,B 0,C 180,E1 -6706.4,E2 -6706.4} C_VEL
LIN {X 0,Y 481.618,Z 111.102,A -85,B 0,C 180,E1 -6706.636,E2 -6706.636} C_VEL
LIN {X 0,Y 481.659,Z 111.109,A -85,B 0,C 180,E1 -6710.058,E2 -6710.058} C_VEL
LIN {X 0,Y 481.622,Z 111.109,A -85,B 0,C 180,E1 -6713.253,E2 -6713.253} C_VEL
LIN {X 0,Y 481.673,Z 111.105,A -85,B 0,C 180,E1 -6716.327,E2 -6716.327} C_VEL
LIN {X 0,Y 481.636,Z 111.108,A -85,B 0,C 180,E1 -6719.421,E2 -6719.421} C_VEL
LIN {X 0,Y 481.652,Z 111.108,A -85,B 0,C 180,E1 -6722.165,E2 -6722.165} C_VEL
LIN {X 0,Y 481.676,Z 111.106,A -85,B 0,C 180,E1 -6724.968,E2 -6724.968} C_VEL
LIN {X 0,Y 481.639,Z 111.112,A -85,B 0,C 180,E1 -6727.704,E2 -6727.704} C_VEL
LIN {X 0,Y 481.696,Z 111.105,A -85,B 0,C 180,E1 -6730.393,E2 -6730.393} C_VEL
LIN {X 0,Y 481.622,Z 111.113,A -85,B 0,C 180,E1 -6733.031,E2 -6733.031} C_VEL
LIN {X 0,Y 481.668,Z 111.109,A -85,B 0,C 180,E1 -6735.638,E2 -6735.638} C_VEL
LIN {X 0,Y 481.755,Z 111.102,A -85,B 0,C 180,E1 -6738.215,E2 -6738.215} C_VEL
LIN {X 0,Y 481.72,Z 111.102,A -85,B 0,C 180,E1 -6741.611,E2 -6741.611} C_VEL
LIN {X 0,Y 481.768,Z 111.101,A -85,B 0,C 180,E1 -6744.139,E2 -6744.139} C_VEL
LIN {X 0,Y 481.909,Z 111.083,A -85,B 0,C 180,E1 -6747.492,E2 -6747.492} C_VEL
LIN {X 0,Y 481.695,Z 111.168,A -85,B 0,C 180,E1 -6749.19,E2 -6749.19} C_VEL
LIN {X 0,Y 483.878,Z 120.467,A -85,B 0,C 180,E1 -6750.624,E2 -6750.624} C_VEL
LIN {X 0,Y 485.307,Z 127.292,A -85,B 0,C 180,E1 -6751.66,E2 -6751.66} C_VEL
LIN {X 0,Y 485.002,Z 141.968,A -85,B 0,C 180,E1 -6753.698,E2 -6753.698} C_VEL
LIN {X 0,Y 488.981,Z 161.032,A -85,B 0,C 180,E1 -6754.197,E2 -6754.197} C_VEL
LIN {X 0,Y 487.422,Z 308.047,A -85,B 0,C 180,E1 -6756.442,E2 -6756.442} C_VEL
LIN {X 0,Y 487.078,Z 322.494,A -85,B 0,C 180,E1 -6756.811,E2 -6756.811} C_VEL
LIN {X 0,Y 486.592,Z 337.493,A -85,B 0,C 180,E1 -6757.365,E2 -6757.365} C_VEL
LIN {X 0,Y 486.002,Z 350.683,A -85,B 0,C 180,E1 -6758.001,E2 -6758.001} C_VEL
LIN {X 0,Y 485.291,Z 364.644,A -85,B 0,C 180,E1 -6758.851,E2 -6758.851} C_VEL
LIN {X 0,Y 484.64,Z 377.462,A -85,B 0,C 180,E1 -6759.817,E2 -6759.817} C_VEL
LIN {X 0,Y 483.801,Z 390.348,A -85,B 0,C 180,E1 -6760.991,E2 -6760.991} C_VEL
LIN {X 0,Y 483.191,Z 401.18,A -85,B 0,C 180,E1 -6762.175,E2 -6762.175} C_VEL
LIN {X 0,Y 482.574,Z 411.213,A -85,B 0,C 180,E1 -6763.475,E2 -6763.475} C_VEL
LIN {X 0,Y 482.026,Z 421.05,A -85,B 0,C 180,E1 -6764.999,E2 -6764.999} C_VEL
LIN {X 0,Y 481.6,Z 429.243,A -85,B 0,C 180,E1 -6766.533,E2 -6766.533} C_VEL
LIN {X 0,Y 481.346,Z 435.097,A -85,B 0,C 180,E1 -6767.855,E2 -6767.855} C_VEL
LIN {X 0,Y 481.069,Z 441.539,A -85,B 0,C 180,E1 -6769.634,E2 -6769.634} C_VEL
LIN {X 0,Y 480.925,Z 446.478,A -85,B 0,C 180,E1 -6771.428,E2 -6771.428} C_VEL
LIN {X 0,Y 480.732,Z 450.025,A -85,B 0,C 180,E1 -6773.249,E2 -6773.249} C_VEL
LIN {X 0,Y 480.675,Z 452.182,A -85,B 0,C 180,E1 -6775.088,E2 -6775.088} C_VEL
LIN {X 0,Y 480.697,Z 452.964,A -85,B 0,C 180,E1 -6776.951,E2 -6776.951} C_VEL
LIN {X 0,Y 480.721,Z 452.327,A -85,B 0,C 180,E1 -6778.846,E2 -6778.846} C_VEL
LIN {X 0,Y 480.798,Z 450.665,A -85,B 0,C 180,E1 -6780.409,E2 -6780.409} C_VEL
LIN {X 0,Y 480.846,Z 447.887,A -85,B 0,C 180,E1 -6782.034,E2 -6782.034} C_VEL
LIN {X 0,Y 481.001,Z 443.777,A -85,B 0,C 180,E1 -6783.726,E2 -6783.726} C_VEL
LIN {X 0,Y 481.185,Z 438.399,A -85,B 0,C 180,E1 -6785.398,E2 -6785.398} C_VEL
LIN {X 0,Y 481.47,Z 431.798,A -85,B 0,C 180,E1 -6787.022,E2 -6787.022} C_VEL
LIN {X 0,Y 481.877,Z 423.858,A -85,B 0,C 180,E1 -6788.61,E2 -6788.61} C_VEL
LIN {X 0,Y 482.37,Z 414.554,A -85,B 0,C 180,E1 -6790.144,E2 -6790.144} C_VEL
LIN {X 0,Y 483.029,Z 403.935,A -85,B 0,C 180,E1 -6791.593,E2 -6791.593} C_VEL
LIN {X 0,Y 483.716,Z 392.125,A -85,B 0,C 180,E1 -6792.934,E2 -6792.934} C_VEL
LIN {X 0,Y 484.432,Z 380.501,A -85,B 0,C 180,E1 -6794.032,E2 -6794.032} C_VEL
LIN {X 0,Y 485.16,Z 367.241,A -85,B 0,C 180,E1 -6795.072,E2 -6795.072} C_VEL
LIN {X 0,Y 485.912,Z 353.632,A -85,B 0,C 180,E1 -6795.937,E2 -6795.937} C_VEL
LIN {X 0,Y 486.469,Z 340.149,A -85,B 0,C 180,E1 -6796.624,E2 -6796.624} C_VEL
LIN {X 0,Y 487.054,Z 325.009,A -85,B 0,C 180,E1 -6797.209,E2 -6797.209} C_VEL
LIN {X 0,Y 487.442,Z 310.61,A -85,B 0,C 180,E1 -6797.602,E2 -6797.602} C_VEL
LIN {X 0,Y 487.671,Z 287.308,A -85,B 0,C 180,E1 -6797.995,E2 -6797.995} C_VEL
LIN {X 0,Y 489.005,Z 156.52,A -85,B 0,C 180,E1 -6799.984,E2 -6799.984} C_VEL
LIN {X 0,Y 486.131,Z 140.508,A -85,B 0,C 180,E1 -6800.395,E2 -6800.395} C_VEL
LIN {X 0,Y 486.357,Z 129.415,A -85,B 0,C 180,E1 -6801.584,E2 -6801.584} C_VEL
LIN {X 0,Y 482.74,Z 115.055,A -85,B 0,C 180,E1 -6803.351,E2 -6803.351} C_VEL
LIN {X 0,Y 481.669,Z 111.113,A -85,B 0,C 180,E1 -6803.873,E2 -6803.873} C_VEL
LIN {X 0,Y 481.713,Z 111.106,A -85,B 0,C 180,E1 -6806.33,E2 -6806.33} C_VEL
LIN {X 0,Y 481.653,Z 111.115,A -85,B 0,C 180,E1 -6809.417,E2 -6809.417} C_VEL
LIN {X 0,Y 481.703,Z 111.107,A -85,B 0,C 180,E1 -6812.168,E2 -6812.168} C_VEL
LIN {X 0,Y 481.72,Z 111.107,A -85,B 0,C 180,E1 -6814.97,E2 -6814.97} C_VEL
LIN {X 0,Y 481.68,Z 111.215,A -85,B 0,C 180,E1 -6816.208,E2 -6816.208} C_VEL
LIN {X 0,Y 482.324,Z 113.756,A -85,B 0,C 180,E1 -6816.586,E2 -6816.586} C_VEL
LIN {X 0,Y 488.907,Z 130.823,A -85,B 0,C 180,E1 -6817.207,E2 -6817.207} C_VEL
LIN {X 0,Y 486.71,Z 280.738,A -85,B 0,C 180,E1 -6819.723,E2 -6819.723} C_VEL
LIN {X 0,Y 486.365,Z 296.263,A -85,B 0,C 180,E1 -6820.15,E2 -6820.15} C_VEL
LIN {X 0,Y 485.886,Z 311.248,A -85,B 0,C 180,E1 -6820.733,E2 -6820.733} C_VEL
LIN {X 0,Y 485.347,Z 324.904,A -85,B 0,C 180,E1 -6821.423,E2 -6821.423} C_VEL
LIN {X 0,Y 484.742,Z 338.369,A -85,B 0,C 180,E1 -6822.274,E2 -6822.274} C_VEL
LIN {X 0,Y 484.146,Z 351.142,A -85,B 0,C 180,E1 -6823.259,E2 -6823.259} C_VEL
LIN {X 0,Y 483.524,Z 363.453,A -85,B 0,C 180,E1 -6824.401,E2 -6824.401} C_VEL
LIN {X 0,Y 482.906,Z 374.924,A -85,B 0,C 180,E1 -6825.675,E2 -6825.675} C_VEL
LIN {X 0,Y 482.335,Z 386.057,A -85,B 0,C 180,E1 -6827.161,E2 -6827.161} C_VEL
LIN {X 0,Y 481.945,Z 395.24,A -85,B 0,C 180,E1 -6828.646,E2 -6828.646} C_VEL
LIN {X 0,Y 481.538,Z 402.837,A -85,B 0,C 180,E1 -6830.125,E2 -6830.125} C_VEL
LIN {X 0,Y 481.317,Z 409.098,A -85,B 0,C 180,E1 -6831.604,E2 -6831.604} C_VEL
LIN {X 0,Y 481.069,Z 415.242,A -85,B 0,C 180,E1 -6833.425,E2 -6833.425} C_VEL
LIN {X 0,Y 480.91,Z 419.176,A -85,B 0,C 180,E1 -6834.969,E2 -6834.969} C_VEL
LIN {X 0,Y 480.981,Z 422.237,A -85,B 0,C 180,E1 -6836.649,E2 -6836.649} C_VEL
LIN {X 0,Y 480.826,Z 424.114,A -85,B 0,C 180,E1 -6838.325,E2 -6838.325} C_VEL
LIN {X 0,Y 480.761,Z 424.807,A -85,B 0,C 180,E1 -6840,E2 -6840} C_VEL
LIN {X 0,Y 480.827,Z 424.283,A -85,B 0,C 180,E1 -6841.675,E2 -6841.675} C_VEL
LIN {X 0,Y 480.994,Z 422.586,A -85,B 0,C 180,E1 -6843.35,E2 -6843.35} C_VEL
LIN {X 0,Y 480.928,Z 419.699,A -85,B 0,C 180,E1 -6845.03,E2 -6845.03} C_VEL
LIN {X 0,Y 481.159,Z 415.52,A -85,B 0,C 180,E1 -6846.71,E2 -6846.71} C_VEL
LIN {X 0,Y 481.36,Z 409.96,A -85,B 0,C 180,E1 -6848.395,E2 -6848.395} C_VEL
LIN {X 0,Y 481.619,Z 402.853,A -85,B 0,C 180,E1 -6850.085,E2 -6850.085} C_VEL
LIN {X 0,Y 482.008,Z 395.191,A -85,B 0,C 180,E1 -6851.565,E2 -6851.565} C_VEL
LIN {X 0,Y 482.397,Z 385.918,A -85,B 0,C 180,E1 -6853.051,E2 -6853.051} C_VEL
LIN {X 0,Y 482.956,Z 376.439,A -85,B 0,C 180,E1 -6854.323,E2 -6854.323} C_VEL
LIN {X 0,Y 483.55,Z 365.136,A -85,B 0,C 180,E1 -6855.598,E2 -6855.598} C_VEL
LIN {X 0,Y 484.219,Z 352.729,A -85,B 0,C 180,E1 -6856.76,E2 -6856.76} C_VEL
LIN {X 0,Y 484.827,Z 338.843,A -85,B 0,C 180,E1 -6857.832,E2 -6857.832} C_VEL
LIN {X 0,Y 485.445,Z 325.236,A -85,B 0,C 180,E1 -6858.682,E2 -6858.682} C_VEL
LIN {X 0,Y 485.951,Z 311.374,A -85,B 0,C 180,E1 -6859.374,E2 -6859.374} C_VEL
LIN {X 0,Y 486.407,Z 296.351,A -85,B 0,C 180,E1 -6859.945,E2 -6859.945} C_VEL
LIN {X 0,Y 486.704,Z 280.878,A -85,B 0,C 180,E1 -6860.36,E2 -6860.36} C_VEL
LIN {X 0,Y 488.619,Z 176.949,A -85,B 0,C 180,E1 -6862.225,E2 -6862.225} C_VEL
LIN {X 0,Y 489.634,Z 133.097,A -85,B 0,C 180,E1 -6863.063,E2 -6863.063} C_VEL
LIN {X 0,Y 485.084,Z 122.538,A -85,B 0,C 180,E1 -6863.579,E2 -6863.579} C_VEL
LIN {X 0,Y 483.872,Z 119.863,A -85,B 0,C 180,E1 -6863.726,E2 -6863.726} C_VEL
LIN {X 0,Y 481.677,Z 111.113,A -85,B 0,C 180,E1 -6865.753,E2 -6865.753} C_VEL
LIN {X 0,Y 481.66,Z 111.114,A -85,B 0,C 180,E1 -6868.784,E2 -6868.784} C_VEL
LIN {X 0,Y 481.642,Z 111.118,A -85,B 0,C 180,E1 -6871.688,E2 -6871.688} C_VEL
LIN {X 0,Y 481.681,Z 111.11,A -85,B 0,C 180,E1 -6874.683,E2 -6874.683} C_VEL
LIN {X 0,Y 481.648,Z 111.114,A -85,B 0,C 180,E1 -6878.006,E2 -6878.006} C_VEL
LIN {X 0,Y 481.622,Z 111.119,A -85,B 0,C 180,E1 -6881.045,E2 -6881.045} C_VEL
LIN {X 0,Y 481.653,Z 111.112,A -85,B 0,C 180,E1 -6884.458,E2 -6884.458} C_VEL
LIN {X 0,Y 481.614,Z 111.121,A -85,B 0,C 180,E1 -6886.855,E2 -6886.855} C_VEL
LIN {X 0,Y 481.656,Z 111.112,A -85,B 0,C 180,E1 -6890.057,E2 -6890.057} C_VEL
LIN {X 0,Y 481.617,Z 111.122,A -85,B 0,C 180,E1 -6893.252,E2 -6893.252} C_VEL
LIN {X 0,Y 481.669,Z 111.114,A -85,B 0,C 180,E1 -6896.327,E2 -6896.327} C_VEL
LIN {X 0,Y 481.65,Z 111.27,A -85,B 0,C 180,E1 -6898.527,E2 -6898.527} C_VEL
LIN {X 0,Y 484.906,Z 123.335,A -85,B 0,C 180,E1 -6900.716,E2 -6900.716} C_VEL
LIN {X 0,Y 486.369,Z 129.906,A -85,B 0,C 180,E1 -6901.817,E2 -6901.817} C_VEL
LIN {X 0,Y 485.466,Z 147.131,A -85,B 0,C 180,E1 -6904.259,E2 -6904.259} C_VEL
LIN {X 0,Y 484.633,Z 162.213,A -85,B 0,C 180,E1 -6906.317,E2 -6906.317} C_VEL
LIN {X 0,Y 487.814,Z 180.405,A -85,B 0,C 180,E1 -6906.897,E2 -6906.897} C_VEL
LIN {X 0,Y 488.944,Z 189.042,A -85,B 0,C 180,E1 -6907.138,E2 -6907.138} C_VEL
LIN {X 0,Y 487.054,Z 288.305,A -85,B 0,C 180,E1 -6908.937,E2 -6908.937} C_VEL
LIN {X 0,Y 486.296,Z 332.214,A -85,B 0,C 180,E1 -6909.705,E2 -6909.705} C_VEL
LIN {X 0,Y 485.791,Z 348.014,A -85,B 0,C 180,E1 -6910.146,E2 -6910.146} C_VEL
LIN {X 0,Y 485.168,Z 366.434,A -85,B 0,C 180,E1 -6910.868,E2 -6910.868} C_VEL
LIN {X 0,Y 484.639,Z 379.124,A -85,B 0,C 180,E1 -6911.505,E2 -6911.505} C_VEL
LIN {X 0,Y 484.043,Z 392.695,A -85,B 0,C 180,E1 -6912.357,E2 -6912.357} C_VEL
LIN {X 0,Y 483.475,Z 405.255,A -85,B 0,C 180,E1 -6913.325,E2 -6913.325} C_VEL
LIN {X 0,Y 482.777,Z 417.748,A -85,B 0,C 180,E1 -6914.485,E2 -6914.485} C_VEL
LIN {X 0,Y 482.336,Z 428.257,A -85,B 0,C 180,E1 -6915.658,E2 -6915.658} C_VEL
LIN {X 0,Y 481.871,Z 437.962,A -85,B 0,C 180,E1 -6916.934,E2 -6916.934} C_VEL
LIN {X 0,Y 481.469,Z 447.454,A -85,B 0,C 180,E1 -6918.422,E2 -6918.422} C_VEL
LIN {X 0,Y 481.216,Z 455.313,A -85,B 0,C 180,E1 -6919.906,E2 -6919.906} C_VEL
LIN {X 0,Y 481.024,Z 462.623,A -85,B 0,C 180,E1 -6921.599,E2 -6921.599} C_VEL
LIN {X 0,Y 480.957,Z 468.418,A -85,B 0,C 180,E1 -6923.287,E2 -6923.287} C_VEL
LIN {X 0,Y 480.876,Z 472.846,A -85,B 0,C 180,E1 -6924.969,E2 -6924.969} C_VEL
LIN {X 0,Y 480.88,Z 475.986,A -85,B 0,C 180,E1 -6926.649,E2 -6926.649} C_VEL
LIN {X 0,Y 480.822,Z 477.87,A -85,B 0,C 180,E1 -6928.325,E2 -6928.325} C_VEL
LIN {X 0,Y 480.751,Z 478.539,A -85,B 0,C 180,E1 -6930,E2 -6930} C_VEL
LIN {X 0,Y 480.822,Z 477.961,A -85,B 0,C 180,E1 -6931.675,E2 -6931.675} C_VEL
LIN {X 0,Y 480.879,Z 476.17,A -85,B 0,C 180,E1 -6933.351,E2 -6933.351} C_VEL
LIN {X 0,Y 480.861,Z 473.139,A -85,B 0,C 180,E1 -6935.031,E2 -6935.031} C_VEL
LIN {X 0,Y 480.969,Z 468.809,A -85,B 0,C 180,E1 -6936.713,E2 -6936.713} C_VEL
LIN {X 0,Y 481.027,Z 463.052,A -85,B 0,C 180,E1 -6938.401,E2 -6938.401} C_VEL
LIN {X 0,Y 481.227,Z 455.726,A -85,B 0,C 180,E1 -6940.093,E2 -6940.093} C_VEL
LIN {X 0,Y 481.528,Z 447.869,A -85,B 0,C 180,E1 -6941.577,E2 -6941.577} C_VEL
LIN {X 0,Y 481.877,Z 438.391,A -85,B 0,C 180,E1 -6943.065,E2 -6943.065} C_VEL
LIN {X 0,Y 482.32,Z 428.748,A -85,B 0,C 180,E1 -6944.342,E2 -6944.342} C_VEL
LIN {X 0,Y 482.936,Z 417.29,A -85,B 0,C 180,E1 -6945.618,E2 -6945.618} C_VEL
LIN {X 0,Y 483.522,Z 404.692,A -85,B 0,C 180,E1 -6946.792,E2 -6946.792} C_VEL
LIN {X 0,Y 484.161,Z 392.316,A -85,B 0,C 180,E1 -6947.748,E2 -6947.748} C_VEL
LIN {X 0,Y 484.864,Z 378.99,A -85,B 0,C 180,E1 -6948.596,E2 -6948.596} C_VEL
LIN {X 0,Y 485.506,Z 364.481,A -85,B 0,C 180,E1 -6949.337,E2 -6949.337} C_VEL
LIN {X 0,Y 486.075,Z 348.943,A -85,B 0,C 180,E1 -6949.942,E2 -6949.942} C_VEL
LIN {X 0,Y 486.526,Z 333.332,A -85,B 0,C 180,E1 -6950.368,E2 -6950.368} C_VEL
LIN {X 0,Y 488.707,Z 185.075,A -85,B 0,C 180,E1 -6952.848,E2 -6952.848} C_VEL
LIN {X 0,Y 485.673,Z 164.191,A -85,B 0,C 180,E1 -6953.373,E2 -6953.373} C_VEL
LIN {X 0,Y 486.657,Z 143.085,A -85,B 0,C 180,E1 -6955.559,E2 -6955.559} C_VEL
LIN {X 0,Y 487.176,Z 131.295,A -85,B 0,C 180,E1 -6956.795,E2 -6956.795} C_VEL
LIN {X 0,Y 481.662,Z 111.116,A -85,B 0,C 180,E1 -6959.32,E2 -6959.32} C_VEL
LIN {X 0,Y 481.65,Z 111.114,A -85,B 0,C 180,E1 -6962.676,E2 -6962.676} C_VEL
LIN {X 0,Y 481.629,Z 111.116,A -85,B 0,C 180,E1 -6965.71,E2 -6965.71} C_VEL
LIN {X 0,Y 481.664,Z 111.113,A -85,B 0,C 180,E1 -6968.86,E2 -6968.86} C_VEL
LIN {X 0,Y 481.614,Z 111.116,A -85,B 0,C 180,E1 -6972.164,E2 -6972.164} C_VEL
LIN {X 0,Y 481.653,Z 111.112,A -85,B 0,C 180,E1 -6974.458,E2 -6974.458} C_VEL
LIN {X 0,Y 481.614,Z 111.118,A -85,B 0,C 180,E1 -6976.855,E2 -6976.855} C_VEL
LIN {X 0,Y 481.656,Z 111.112,A -85,B 0,C 180,E1 -6980.058,E2 -6980.058} C_VEL
LIN {X 0,Y 481.619,Z 111.117,A -85,B 0,C 180,E1 -6983.253,E2 -6983.253} C_VEL
LIN {X 0,Y 481.67,Z 111.114,A -85,B 0,C 180,E1 -6986.327,E2 -6986.327} C_VEL
LIN {X 0,Y 481.645,Z 111.113,A -85,B 0,C 180,E1 -6989.419,E2 -6989.419} C_VEL
LIN {X 0,Y 481.651,Z 111.116,A -85,B 0,C 180,E1 -6992.165,E2 -6992.165} C_VEL
LIN {X 0,Y 481.682,Z 111.274,A -85,B 0,C 180,E1 -6995.285,E2 -6995.285} C_VEL
LIN {X 0,Y 483.559,Z 118.028,A -85,B 0,C 180,E1 -6996.356,E2 -6996.356} C_VEL
LIN {X 0,Y 488.552,Z 129.604,A -85,B 0,C 180,E1 -6996.927,E2 -6996.927} C_VEL
LIN {X 0,Y 489.561,Z 132.834,A -85,B 0,C 180,E1 -6997.054,E2 -6997.054} C_VEL
LIN {X 0,Y 487.493,Z 226.464,A -85,B 0,C 180,E1 -6998.791,E2 -6998.791} C_VEL
LIN {X 0,Y 486.625,Z 282.857,A -85,B 0,C 180,E1 -6999.791,E2 -6999.791} C_VEL
LIN {X 0,Y 486.259,Z 298.479,A -85,B 0,C 180,E1 -7000.232,E2 -7000.232} C_VEL
LIN {X 0,Y 485.818,Z 313.73,A -85,B 0,C 180,E1 -7000.84,E2 -7000.84} C_VEL
LIN {X 0,Y 485.336,Z 327.051,A -85,B 0,C 180,E1 -7001.533,E2 -7001.533} C_VEL
LIN {X 0,Y 484.729,Z 340.291,A -85,B 0,C 180,E1 -7002.383,E2 -7002.383} C_VEL
LIN {X 0,Y 484.086,Z 352.993,A -85,B 0,C 180,E1 -7003.374,E2 -7003.374} C_VEL
LIN {X 0,Y 483.473,Z 365.037,A -85,B 0,C 180,E1 -7004.508,E2 -7004.508} C_VEL
LIN {X 0,Y 482.959,Z 375.458,A -85,B 0,C 180,E1 -7005.678,E2 -7005.678} C_VEL
LIN {X 0,Y 482.479,Z 385.092,A -85,B 0,C 180,E1 -7006.951,E2 -7006.951} C_VEL
LIN {X 0,Y 482.053,Z 393.278,A -85,B 0,C 180,E1 -7008.223,E2 -7008.223} C_VEL
LIN {X 0,Y 481.669,Z 401.273,A -85,B 0,C 180,E1 -7009.704,E2 -7009.704} C_VEL
LIN {X 0,Y 481.4,Z 407.859,A -85,B 0,C 180,E1 -7011.183,E2 -7011.183} C_VEL
LIN {X 0,Y 481.172,Z 413.888,A -85,B 0,C 180,E1 -7012.869,E2 -7012.869} C_VEL
LIN {X 0,Y 481.115,Z 417.419,A -85,B 0,C 180,E1 -7014.131,E2 -7014.131} C_VEL
LIN {X 0,Y 480.995,Z 421.02,A -85,B 0,C 180,E1 -7015.811,E2 -7015.811} C_VEL
LIN {X 0,Y 480.944,Z 423.381,A -85,B 0,C 180,E1 -7017.488,E2 -7017.488} C_VEL
LIN {X 0,Y 480.77,Z 424.563,A -85,B 0,C 180,E1 -7019.163,E2 -7019.163} C_VEL
LIN {X 0,Y 480.77,Z 424.527,A -85,B 0,C 180,E1 -7020.838,E2 -7020.838} C_VEL
LIN {X 0,Y 480.943,Z 423.309,A -85,B 0,C 180,E1 -7022.513,E2 -7022.513} C_VEL
LIN {X 0,Y 480.972,Z 420.917,A -85,B 0,C 180,E1 -7024.19,E2 -7024.19} C_VEL
LIN {X 0,Y 481.09,Z 417.285,A -85,B 0,C 180,E1 -7025.87,E2 -7025.87} C_VEL
LIN {X 0,Y 481.185,Z 412.335,A -85,B 0,C 180,E1 -7027.554,E2 -7027.554} C_VEL
LIN {X 0,Y 481.408,Z 405.931,A -85,B 0,C 180,E1 -7029.241,E2 -7029.241} C_VEL
LIN {X 0,Y 481.788,Z 397.877,A -85,B 0,C 180,E1 -7030.932,E2 -7030.932} C_VEL
LIN {X 0,Y 482.075,Z 389.527,A -85,B 0,C 180,E1 -7032.374,E2 -7032.374} C_VEL
LIN {X 0,Y 482.602,Z 380.455,A -85,B 0,C 180,E1 -7033.689,E2 -7033.689} C_VEL
LIN {X 0,Y 483.148,Z 370.064,A -85,B 0,C 180,E1 -7034.963,E2 -7034.963} C_VEL
LIN {X 0,Y 483.79,Z 357.925,A -85,B 0,C 180,E1 -7036.208,E2 -7036.208} C_VEL
LIN {X 0,Y 484.41,Z 345.086,A -85,B 0,C 180,E1 -7037.303,E2 -7037.303} C_VEL
LIN {X 0,Y 485.057,Z 331.4,A -85,B 0,C 180,E1 -7038.26,E2 -7038.26} C_VEL
LIN {X 0,Y 485.632,Z 317.216,A -85,B 0,C 180,E1 -7039.058,E2 -7039.058} C_VEL
LIN {X 0,Y 486.164,Z 301.713,A -85,B 0,C 180,E1 -7039.733,E2 -7039.733} C_VEL
LIN {X 0,Y 486.561,Z 286.838,A -85,B 0,C 180,E1 -7040.205,E2 -7040.205} C_VEL
LIN {X 0,Y 486.81,Z 270.43,A -85,B 0,C 180,E1 -7040.549,E2 -7040.549} C_VEL
LIN {X 0,Y 488.828,Z 133.292,A -85,B 0,C 180,E1 -7042.822,E2 -7042.822} C_VEL
LIN {X 0,Y 487.818,Z 128.684,A -85,B 0,C 180,E1 -7042.952,E2 -7042.952} C_VEL
LIN {X 0,Y 482.412,Z 114.39,A -85,B 0,C 180,E1 -7043.486,E2 -7043.486} C_VEL
LIN {X 0,Y 481.657,Z 111.115,A -85,B 0,C 180,E1 -7044.063,E2 -7044.063} C_VEL
LIN {X 0,Y 481.685,Z 111.108,A -85,B 0,C 180,E1 -7047.124,E2 -7047.124} C_VEL
LIN {X 0,Y 481.668,Z 111.115,A -85,B 0,C 180,E1 -7049.742,E2 -7049.742} C_VEL
LIN {X 0,Y 481.654,Z 111.11,A -85,B 0,C 180,E1 -7052.676,E2 -7052.676} C_VEL
LIN {X 0,Y 481.632,Z 111.118,A -85,B 0,C 180,E1 -7055.71,E2 -7055.71} C_VEL
LIN {X 0,Y 481.668,Z 111.109,A -85,B 0,C 180,E1 -7058.86,E2 -7058.86} C_VEL
LIN {X 0,Y 481.626,Z 111.113,A -85,B 0,C 180,E1 -7062.164,E2 -7062.164} C_VEL
LIN {X 0,Y 481.656,Z 111.101,A -85,B 0,C 180,E1 -7065.542,E2 -7065.542} C_VEL
LIN {X 0,Y 481.618,Z 111.102,A -85,B 0,C 180,E1 -7066.636,E2 -7066.636} C_VEL
LIN {X 0,Y 480.967,Z 111.19,A -85,B 0,C 180,E1 -7067.334,E2 -7067.334} C_VEL
LIN {X 0,Y 478.095,Z 111.549,A -85,B 0,C 180,E1 -7068.469,E2 -7068.469} C_VEL
LIN {X 0,Y 475.676,Z 111.86,A -85,B 0,C 180,E1 -7069.383,E2 -7069.383} C_VEL
LIN {X 0,Y 474.668,Z 111.98,A -85,B 0,C 180,E1 -7070.09,E2 -7070.09} C_VEL
LIN {X 0,Y 474.604,Z 111.988,A -85,B 0,C 180,E1 -7070.329,E2 -7070.329} C_VEL
LIN {X 0,Y 474.568,Z 111.99,A -85,B 0,C 180,E1 -7073.102,E2 -7073.102} C_VEL
LIN {X 0,Y 474.623,Z 111.982,A -85,B 0,C 180,E1 -7076.02,E2 -7076.02} C_VEL
LIN {X 0,Y 474.592,Z 111.995,A -85,B 0,C 180,E1 -7078.782,E2 -7078.782} C_VEL
LIN {X 0,Y 474.604,Z 111.986,A -85,B 0,C 180,E1 -7081.715,E2 -7081.715} C_VEL
LIN {X 0,Y 474.612,Z 111.992,A -85,B 0,C 180,E1 -7084.594,E2 -7084.594} C_VEL
LIN {X 0,Y 474.587,Z 111.991,A -85,B 0,C 180,E1 -7087.355,E2 -7087.355} C_VEL
LIN {X 0,Y 474.645,Z 111.981,A -85,B 0,C 180,E1 -7090.089,E2 -7090.089} C_VEL
LIN {X 0,Y 474.596,Z 111.992,A -85,B 0,C 180,E1 -7092.772,E2 -7092.772} C_VEL
LIN {X 0,Y 474.629,Z 111.986,A -85,B 0,C 180,E1 -7095.42,E2 -7095.42} C_VEL
LIN {X 0,Y 474.708,Z 111.978,A -85,B 0,C 180,E1 -7098.038,E2 -7098.038} C_VEL
LIN {X 0,Y 474.669,Z 111.98,A -85,B 0,C 180,E1 -7101.485,E2 -7101.485} C_VEL
LIN {X 0,Y 474.731,Z 111.977,A -85,B 0,C 180,E1 -7104.052,E2 -7104.052} C_VEL
LIN {X 0,Y 474.874,Z 111.96,A -85,B 0,C 180,E1 -7107.455,E2 -7107.455} C_VEL
LIN {X 0,Y 474.691,Z 112.149,A -85,B 0,C 180,E1 -7108.913,E2 -7108.913} C_VEL
LIN {X 0,Y 476.983,Z 121.824,A -85,B 0,C 180,E1 -7110.422,E2 -7110.422} C_VEL
LIN {X 0,Y 478.449,Z 128.652,A -85,B 0,C 180,E1 -7111.472,E2 -7111.472} C_VEL
LIN {X 0,Y 478.204,Z 141.996,A -85,B 0,C 180,E1 -7113.344,E2 -7113.344} C_VEL
LIN {X 0,Y 482.431,Z 161.937,A -85,B 0,C 180,E1 -7113.889,E2 -7113.889} C_VEL
LIN {X 0,Y 480.756,Z 308.205,A -85,B 0,C 180,E1 -7116.152,E2 -7116.152} C_VEL
LIN {X 0,Y 480.393,Z 323.305,A -85,B 0,C 180,E1 -7116.548,E2 -7116.548} C_VEL
LIN {X 0,Y 479.867,Z 337.918,A -85,B 0,C 180,E1 -7117.098,E2 -7117.098} C_VEL
LIN {X 0,Y 479.224,Z 351.985,A -85,B 0,C 180,E1 -7117.796,E2 -7117.796} C_VEL
LIN {X 0,Y 478.464,Z 365.743,A -85,B 0,C 180,E1 -7118.659,E2 -7118.659} C_VEL
LIN {X 0,Y 477.776,Z 377.713,A -85,B 0,C 180,E1 -7119.576,E2 -7119.576} C_VEL
LIN {X 0,Y 476.969,Z 390.142,A -85,B 0,C 180,E1 -7120.721,E2 -7120.721} C_VEL
LIN {X 0,Y 476.295,Z 401.032,A -85,B 0,C 180,E1 -7121.922,E2 -7121.922} C_VEL
LIN {X 0,Y 475.663,Z 410.788,A -85,B 0,C 180,E1 -7123.196,E2 -7123.196} C_VEL
LIN {X 0,Y 475.051,Z 421.003,A -85,B 0,C 180,E1 -7124.785,E2 -7124.785} C_VEL
LIN {X 0,Y 474.526,Z 430.268,A -85,B 0,C 180,E1 -7126.565,E2 -7126.565} C_VEL
LIN {X 0,Y 474.228,Z 436.911,A -85,B 0,C 180,E1 -7128.133,E2 -7128.133} C_VEL
LIN {X 0,Y 473.946,Z 442.984,A -85,B 0,C 180,E1 -7129.941,E2 -7129.941} C_VEL
LIN {X 0,Y 473.78,Z 447.591,A -85,B 0,C 180,E1 -7131.768,E2 -7131.768} C_VEL
LIN {X 0,Y 473.612,Z 450.812,A -85,B 0,C 180,E1 -7133.619,E2 -7133.619} C_VEL
LIN {X 0,Y 473.581,Z 452.65,A -85,B 0,C 180,E1 -7135.491,E2 -7135.491} C_VEL
LIN {X 0,Y 473.586,Z 453.106,A -85,B 0,C 180,E1 -7137.39,E2 -7137.39} C_VEL
LIN {X 0,Y 473.623,Z 452.497,A -85,B 0,C 180,E1 -7138.896,E2 -7138.896} C_VEL
LIN {X 0,Y 473.702,Z 450.642,A -85,B 0,C 180,E1 -7140.626,E2 -7140.626} C_VEL
LIN {X 0,Y 473.806,Z 446.635,A -85,B 0,C 180,E1 -7142.78,E2 -7142.78} C_VEL
LIN {X 0,Y 473.958,Z 442.648,A -85,B 0,C 180,E1 -7144.297,E2 -7144.297} C_VEL
LIN {X 0,Y 474.236,Z 436.505,A -85,B 0,C 180,E1 -7146.092,E2 -7146.092} C_VEL
LIN {X 0,Y 474.625,Z 428.833,A -85,B 0,C 180,E1 -7147.853,E2 -7147.853} C_VEL
LIN {X 0,Y 475.084,Z 419.971,A -85,B 0,C 180,E1 -7149.502,E2 -7149.502} C_VEL
LIN {X 0,Y 475.657,Z 411.386,A -85,B 0,C 180,E1 -7150.837,E2 -7150.837} C_VEL
LIN {X 0,Y 476.328,Z 401.232,A -85,B 0,C 180,E1 -7152.17,E2 -7152.17} C_VEL
LIN {X 0,Y 476.992,Z 390.197,A -85,B 0,C 180,E1 -7153.391,E2 -7153.391} C_VEL
LIN {X 0,Y 477.865,Z 377.223,A -85,B 0,C 180,E1 -7154.579,E2 -7154.579} C_VEL
LIN {X 0,Y 478.564,Z 365.016,A -85,B 0,C 180,E1 -7155.508,E2 -7155.508} C_VEL
LIN {X 0,Y 479.287,Z 351.54,A -85,B 0,C 180,E1 -7156.345,E2 -7156.345} C_VEL
LIN {X 0,Y 479.95,Z 336.771,A -85,B 0,C 180,E1 -7157.068,E2 -7157.068} C_VEL
LIN {X 0,Y 480.465,Z 321.132,A -85,B 0,C 180,E1 -7157.633,E2 -7157.633} C_VEL
LIN {X 0,Y 480.848,Z 306.11,A -85,B 0,C 180,E1 -7158,E2 -7158} C_VEL
LIN {X 0,Y 482.468,Z 157.183,A -85,B 0,C 180,E1 -7160.307,E2 -7160.307} C_VEL
LIN {X 0,Y 479.418,Z 140.51,A -85,B 0,C 180,E1 -7160.754,E2 -7160.754} C_VEL
LIN {X 0,Y 479.662,Z 131.275,A -85,B 0,C 180,E1 -7161.765,E2 -7161.765} C_VEL
LIN {X 0,Y 475.498,Z 115.263,A -85,B 0,C 180,E1 -7163.756,E2 -7163.756} C_VEL
LIN {X 0,Y 474.619,Z 111.992,A -85,B 0,C 180,E1 -7164.175,E2 -7164.175} C_VEL
LIN {X 0,Y 474.646,Z 111.986,A -85,B 0,C 180,E1 -7166.78,E2 -7166.78} C_VEL
LIN {X 0,Y 474.608,Z 111.992,A -85,B 0,C 180,E1 -7169.77,E2 -7169.77} C_VEL
LIN {X 0,Y 474.7,Z 111.979,A -85,B 0,C 180,E1 -7172.68,E2 -7172.68} C_VEL
LIN {X 0,Y 474.656,Z 112.107,A -85,B 0,C 180,E1 -7175.942,E2 -7175.942} C_VEL
LIN {X 0,Y 475.135,Z 114.137,A -85,B 0,C 180,E1 -7176.236,E2 -7176.236} C_VEL
LIN {X 0,Y 482.274,Z 132.057,A -85,B 0,C 180,E1 -7176.914,E2 -7176.914} C_VEL
LIN {X 0,Y 479.962,Z 281.248,A -85,B 0,C 180,E1 -7179.475,E2 -7179.475} C_VEL
LIN {X 0,Y 479.585,Z 296.988,A -85,B 0,C 180,E1 -7179.919,E2 -7179.919} C_VEL
LIN {X 0,Y 479.085,Z 311.752,A -85,B 0,C 180,E1 -7180.504,E2 -7180.504} C_VEL
LIN {X 0,Y 478.478,Z 326.278,A -85,B 0,C 180,E1 -7181.258,E2 -7181.258} C_VEL
LIN {X 0,Y 477.846,Z 339.591,A -85,B 0,C 180,E1 -7182.12,E2 -7182.12} C_VEL
LIN {X 0,Y 477.121,Z 353.463,A -85,B 0,C 180,E1 -7183.226,E2 -7183.226} C_VEL
LIN {X 0,Y 476.547,Z 365.457,A -85,B 0,C 180,E1 -7184.386,E2 -7184.386} C_VEL
LIN {X 0,Y 475.906,Z 376.676,A -85,B 0,C 180,E1 -7185.678,E2 -7185.678} C_VEL
LIN {X 0,Y 475.354,Z 386.137,A -85,B 0,C 180,E1 -7186.969,E2 -7186.969} C_VEL
LIN {X 0,Y 474.923,Z 395.382,A -85,B 0,C 180,E1 -7188.476,E2 -7188.476} C_VEL
LIN {X 0,Y 474.493,Z 403.037,A -85,B 0,C 180,E1 -7189.977,E2 -7189.977} C_VEL
LIN {X 0,Y 474.265,Z 409.348,A -85,B 0,C 180,E1 -7191.478,E2 -7191.478} C_VEL
LIN {X 0,Y 474.019,Z 415.127,A -85,B 0,C 180,E1 -7193.188,E2 -7193.188} C_VEL
LIN {X 0,Y 473.947,Z 418.574,A -85,B 0,C 180,E1 -7194.469,E2 -7194.469} C_VEL
LIN {X 0,Y 473.897,Z 421.208,A -85,B 0,C 180,E1 -7195.747,E2 -7195.747} C_VEL
LIN {X 0,Y 473.885,Z 423.695,A -85,B 0,C 180,E1 -7197.45,E2 -7197.45} C_VEL
LIN {X 0,Y 473.699,Z 425.008,A -85,B 0,C 180,E1 -7199.15,E2 -7199.15} C_VEL
LIN {X 0,Y 473.701,Z 425.098,A -85,B 0,C 180,E1 -7200.85,E2 -7200.85} C_VEL
LIN {X 0,Y 473.887,Z 423.993,A -85,B 0,C 180,E1 -7202.55,E2 -7202.55} C_VEL
LIN {X 0,Y 473.941,Z 421.709,A -85,B 0,C 180,E1 -7204.252,E2 -7204.252} C_VEL
LIN {X 0,Y 474.069,Z 418.181,A -85,B 0,C 180,E1 -7205.956,E2 -7205.956} C_VEL
LIN {X 0,Y 474.189,Z 413.331,A -85,B 0,C 180,E1 -7207.665,E2 -7207.665} C_VEL
LIN {X 0,Y 474.447,Z 407.013,A -85,B 0,C 180,E1 -7209.378,E2 -7209.378} C_VEL
LIN {X 0,Y 474.838,Z 399.028,A -85,B 0,C 180,E1 -7211.093,E2 -7211.093} C_VEL
LIN {X 0,Y 475.205,Z 390.775,A -85,B 0,C 180,E1 -7212.551,E2 -7212.551} C_VEL
LIN {X 0,Y 475.813,Z 381.73,A -85,B 0,C 180,E1 -7213.888,E2 -7213.888} C_VEL
LIN {X 0,Y 476.381,Z 371.38,A -85,B 0,C 180,E1 -7215.18,E2 -7215.18} C_VEL
LIN {X 0,Y 477.079,Z 359.273,A -85,B 0,C 180,E1 -7216.441,E2 -7216.441} C_VEL
LIN {X 0,Y 477.725,Z 346.415,A -85,B 0,C 180,E1 -7217.552,E2 -7217.552} C_VEL
LIN {X 0,Y 478.411,Z 332.701,A -85,B 0,C 180,E1 -7218.522,E2 -7218.522} C_VEL
LIN {X 0,Y 478.988,Z 318.467,A -85,B 0,C 180,E1 -7219.332,E2 -7219.332} C_VEL
LIN {X 0,Y 479.522,Z 303.171,A -85,B 0,C 180,E1 -7220.003,E2 -7220.003} C_VEL
LIN {X 0,Y 479.947,Z 287.108,A -85,B 0,C 180,E1 -7220.513,E2 -7220.513} C_VEL
LIN {X 0,Y 480.29,Z 265.253,A -85,B 0,C 180,E1 -7220.952,E2 -7220.952} C_VEL
LIN {X 0,Y 482.206,Z 178.078,A -85,B 0,C 180,E1 -7222.565,E2 -7222.565} C_VEL
LIN {X 0,Y 483.307,Z 134.813,A -85,B 0,C 180,E1 -7223.424,E2 -7223.424} C_VEL
LIN {X 0,Y 477.915,Z 122.958,A -85,B 0,C 180,E1 -7224.051,E2 -7224.051} C_VEL
LIN {X 0,Y 476.877,Z 120.687,A -85,B 0,C 180,E1 -7224.179,E2 -7224.179} C_VEL
LIN {X 0,Y 474.609,Z 111.994,A -85,B 0,C 180,E1 -7226.256,E2 -7226.256} C_VEL
LIN {X 0,Y 474.6,Z 111.994,A -85,B 0,C 180,E1 -7229.253,E2 -7229.253} C_VEL
LIN {X 0,Y 474.601,Z 111.992,A -85,B 0,C 180,E1 -7232.428,E2 -7232.428} C_VEL
LIN {X 0,Y 474.609,Z 111.994,A -85,B 0,C 180,E1 -7235.468,E2 -7235.468} C_VEL
LIN {X 0,Y 474.608,Z 111.99,A -85,B 0,C 180,E1 -7238.457,E2 -7238.457} C_VEL
LIN {X 0,Y 474.591,Z 111.995,A -85,B 0,C 180,E1 -7241.788,E2 -7241.788} C_VEL
LIN {X 0,Y 474.615,Z 111.991,A -85,B 0,C 180,E1 -7244.702,E2 -7244.702} C_VEL
LIN {X 0,Y 474.575,Z 111.995,A -85,B 0,C 180,E1 -7247.77,E2 -7247.77} C_VEL
LIN {X 0,Y 474.621,Z 111.99,A -85,B 0,C 180,E1 -7250.452,E2 -7250.452} C_VEL
LIN {X 0,Y 474.581,Z 111.996,A -85,B 0,C 180,E1 -7253.676,E2 -7253.676} C_VEL
LIN {X 0,Y 474.612,Z 111.994,A -85,B 0,C 180,E1 -7256.777,E2 -7256.777} C_VEL
LIN {X 0,Y 474.618,Z 112.047,A -85,B 0,C 180,E1 -7258.005,E2 -7258.005} C_VEL
LIN {X 0,Y 477.805,Z 123.619,A -85,B 0,C 180,E1 -7260.207,E2 -7260.207} C_VEL
LIN {X 0,Y 479.727,Z 132.741,A -85,B 0,C 180,E1 -7261.773,E2 -7261.773} C_VEL
LIN {X 0,Y 478.443,Z 152.085,A -85,B 0,C 180,E1 -7264.554,E2 -7264.554} C_VEL
LIN {X 0,Y 477.905,Z 161.8,A -85,B 0,C 180,E1 -7265.894,E2 -7265.894} C_VEL
LIN {X 0,Y 481.274,Z 180.398,A -85,B 0,C 180,E1 -7266.509,E2 -7266.509} C_VEL
LIN {X 0,Y 482.53,Z 190.046,A -85,B 0,C 180,E1 -7266.793,E2 -7266.793} C_VEL
LIN {X 0,Y 480.46,Z 286.783,A -85,B 0,C 180,E1 -7268.606,E2 -7268.606} C_VEL
LIN {X 0,Y 479.601,Z 332.406,A -85,B 0,C 180,E1 -7269.433,E2 -7269.433} C_VEL
LIN {X 0,Y 479.014,Z 348.545,A -85,B 0,C 180,E1 -7269.902,E2 -7269.902} C_VEL
LIN {X 0,Y 478.478,Z 365.101,A -85,B 0,C 180,E1 -7270.534,E2 -7270.534} C_VEL
LIN {X 0,Y 477.858,Z 378.969,A -85,B 0,C 180,E1 -7271.233,E2 -7271.233} C_VEL
LIN {X 0,Y 477.222,Z 392.527,A -85,B 0,C 180,E1 -7272.096,E2 -7272.096} C_VEL
LIN {X 0,Y 476.595,Z 404.973,A -85,B 0,C 180,E1 -7273.068,E2 -7273.068} C_VEL
LIN {X 0,Y 475.882,Z 417.561,A -85,B 0,C 180,E1 -7274.254,E2 -7274.254} C_VEL
LIN {X 0,Y 475.386,Z 428.068,A -85,B 0,C 180,E1 -7275.444,E2 -7275.444} C_VEL
LIN {X 0,Y 474.902,Z 437.773,A -85,B 0,C 180,E1 -7276.739,E2 -7276.739} C_VEL
LIN {X 0,Y 474.405,Z 447.253,A -85,B 0,C 180,E1 -7278.247,E2 -7278.247} C_VEL
LIN {X 0,Y 474.174,Z 455.108,A -85,B 0,C 180,E1 -7279.755,E2 -7279.755} C_VEL
LIN {X 0,Y 473.934,Z 462.406,A -85,B 0,C 180,E1 -7281.472,E2 -7281.472} C_VEL
LIN {X 0,Y 473.887,Z 468.151,A -85,B 0,C 180,E1 -7283.186,E2 -7283.186} C_VEL
LIN {X 0,Y 473.81,Z 472.484,A -85,B 0,C 180,E1 -7284.894,E2 -7284.894} C_VEL
LIN {X 0,Y 473.806,Z 475.575,A -85,B 0,C 180,E1 -7286.599,E2 -7286.599} C_VEL
LIN {X 0,Y 473.756,Z 477.467,A -85,B 0,C 180,E1 -7288.3,E2 -7288.3} C_VEL
LIN {X 0,Y 473.677,Z 478.143,A -85,B 0,C 180,E1 -7290,E2 -7290} C_VEL
LIN {X 0,Y 473.755,Z 477.567,A -85,B 0,C 180,E1 -7291.7,E2 -7291.7} C_VEL
LIN {X 0,Y 473.805,Z 475.767,A -85,B 0,C 180,E1 -7293.401,E2 -7293.401} C_VEL
LIN {X 0,Y 473.789,Z 472.721,A -85,B 0,C 180,E1 -7295.106,E2 -7295.106} C_VEL
LIN {X 0,Y 473.892,Z 468.368,A -85,B 0,C 180,E1 -7296.814,E2 -7296.814} C_VEL
LIN {X 0,Y 473.938,Z 462.581,A -85,B 0,C 180,E1 -7298.528,E2 -7298.528} C_VEL
LIN {X 0,Y 474.197,Z 455.23,A -85,B 0,C 180,E1 -7300.245,E2 -7300.245} C_VEL
LIN {X 0,Y 474.45,Z 447.375,A -85,B 0,C 180,E1 -7301.752,E2 -7301.752} C_VEL
LIN {X 0,Y 474.863,Z 437.891,A -85,B 0,C 180,E1 -7303.262,E2 -7303.262} C_VEL
LIN {X 0,Y 475.33,Z 428.153,A -85,B 0,C 180,E1 -7304.558,E2 -7304.558} C_VEL
LIN {X 0,Y 475.961,Z 416.56,A -85,B 0,C 180,E1 -7305.853,E2 -7305.853} C_VEL
LIN {X 0,Y 476.615,Z 403.818,A -85,B 0,C 180,E1 -7307.042,E2 -7307.042} C_VEL
LIN {X 0,Y 477.415,Z 389.81,A -85,B 0,C 180,E1 -7308.118,E2 -7308.118} C_VEL
LIN {X 0,Y 478.112,Z 375.978,A -85,B 0,C 180,E1 -7308.979,E2 -7308.979} C_VEL
LIN {X 0,Y 478.806,Z 362.001,A -85,B 0,C 180,E1 -7309.675,E2 -7309.675} C_VEL
LIN {X 0,Y 479.351,Z 347.321,A -85,B 0,C 180,E1 -7310.235,E2 -7310.235} C_VEL
LIN {X 0,Y 479.771,Z 332.397,A -85,B 0,C 180,E1 -7310.639,E2 -7310.639} C_VEL
LIN {X 0,Y 482.082,Z 185.401,A -85,B 0,C 180,E1 -7313.151,E2 -7313.151} C_VEL
LIN {X 0,Y 478.935,Z 163.794,A -85,B 0,C 180,E1 -7313.717,E2 -7313.717} C_VEL
LIN {X 0,Y 480.401,Z 135.777,A -85,B 0,C 180,E1 -7316.662,E2 -7316.662} C_VEL
LIN {X 0,Y 480.376,Z 132.946,A -85,B 0,C 180,E1 -7316.971,E2 -7316.971} C_VEL
LIN {X 0,Y 474.626,Z 111.991,A -85,B 0,C 180,E1 -7319.616,E2 -7319.616} C_VEL
LIN {X 0,Y 474.599,Z 111.992,A -85,B 0,C 180,E1 -7322.428,E2 -7322.428} C_VEL
LIN {X 0,Y 474.608,Z 111.991,A -85,B 0,C 180,E1 -7325.468,E2 -7325.468} C_VEL
LIN {X 0,Y 474.607,Z 111.992,A -85,B 0,C 180,E1 -7328.458,E2 -7328.458} C_VEL
LIN {X 0,Y 474.591,Z 111.991,A -85,B 0,C 180,E1 -7331.789,E2 -7331.789} C_VEL
LIN {X 0,Y 474.615,Z 111.991,A -85,B 0,C 180,E1 -7334.702,E2 -7334.702} C_VEL
LIN {X 0,Y 474.575,Z 111.991,A -85,B 0,C 180,E1 -7337.77,E2 -7337.77} C_VEL
LIN {X 0,Y 474.621,Z 111.991,A -85,B 0,C 180,E1 -7340.452,E2 -7340.452} C_VEL
LIN {X 0,Y 474.583,Z 111.993,A -85,B 0,C 180,E1 -7343.676,E2 -7343.676} C_VEL
LIN {X 0,Y 474.614,Z 111.991,A -85,B 0,C 180,E1 -7346.778,E2 -7346.778} C_VEL
LIN {X 0,Y 474.597,Z 111.992,A -85,B 0,C 180,E1 -7349.769,E2 -7349.769} C_VEL
LIN {X 0,Y 474.637,Z 111.989,A -85,B 0,C 180,E1 -7352.676,E2 -7352.676} C_VEL
LIN {X 0,Y 474.671,Z 112.153,A -85,B 0,C 180,E1 -7354.847,E2 -7354.847} C_VEL
LIN {X 0,Y 476.476,Z 118.541,A -85,B 0,C 180,E1 -7355.89,E2 -7355.89} C_VEL
LIN {X 0,Y 482.281,Z 131.545,A -85,B 0,C 180,E1 -7356.574,E2 -7356.574} C_VEL
LIN {X 0,Y 483.297,Z 135.128,A -85,B 0,C 180,E1 -7356.717,E2 -7356.717} C_VEL
LIN {X 0,Y 480.779,Z 235.169,A -85,B 0,C 180,E1 -7358.621,E2 -7358.621} C_VEL
LIN {X 0,Y 479.974,Z 283.713,A -85,B 0,C 180,E1 -7359.511,E2 -7359.511} C_VEL
LIN {X 0,Y 479.581,Z 298.987,A -85,B 0,C 180,E1 -7359.953,E2 -7359.953} C_VEL
LIN {X 0,Y 479.115,Z 314,A -85,B 0,C 180,E1 -7360.562,E2 -7360.562} C_VEL
LIN {X 0,Y 478.605,Z 327.323,A -85,B 0,C 180,E1 -7361.264,E2 -7361.264} C_VEL
LIN {X 0,Y 477.971,Z 340.569,A -85,B 0,C 180,E1 -7362.125,E2 -7362.125} C_VEL
LIN {X 0,Y 477.252,Z 353.811,A -85,B 0,C 180,E1 -7363.174,E2 -7363.174} C_VEL
LIN {X 0,Y 476.61,Z 365.353,A -85,B 0,C 180,E1 -7364.279,E2 -7364.279} C_VEL
LIN {X 0,Y 476.059,Z 375.791,A -85,B 0,C 180,E1 -7365.465,E2 -7365.465} C_VEL
LIN {X 0,Y 475.534,Z 385.445,A -85,B 0,C 180,E1 -7366.757,E2 -7366.757} C_VEL
LIN {X 0,Y 475.049,Z 394.855,A -85,B 0,C 180,E1 -7368.263,E2 -7368.263} C_VEL
LIN {X 0,Y 474.632,Z 402.643,A -85,B 0,C 180,E1 -7369.765,E2 -7369.765} C_VEL
LIN {X 0,Y 474.312,Z 409.865,A -85,B 0,C 180,E1 -7371.479,E2 -7371.479} C_VEL
LIN {X 0,Y 474.062,Z 415.528,A -85,B 0,C 180,E1 -7373.189,E2 -7373.189} C_VEL
LIN {X 0,Y 474.063,Z 417.819,A -85,B 0,C 180,E1 -7374.044,E2 -7374.044} C_VEL
LIN {X 0,Y 473.915,Z 421.423,A -85,B 0,C 180,E1 -7375.748,E2 -7375.748} C_VEL
LIN {X 0,Y 473.885,Z 423.782,A -85,B 0,C 180,E1 -7377.45,E2 -7377.45} C_VEL
LIN {X 0,Y 473.698,Z 424.957,A -85,B 0,C 180,E1 -7379.15,E2 -7379.15} C_VEL
LIN {X 0,Y 473.698,Z 424.909,A -85,B 0,C 180,E1 -7380.85,E2 -7380.85} C_VEL
LIN {X 0,Y 473.867,Z 423.671,A -85,B 0,C 180,E1 -7382.55,E2 -7382.55} C_VEL
LIN {X 0,Y 473.879,Z 421.254,A -85,B 0,C 180,E1 -7384.253,E2 -7384.253} C_VEL
LIN {X 0,Y 474.033,Z 417.588,A -85,B 0,C 180,E1 -7385.957,E2 -7385.957} C_VEL
LIN {X 0,Y 474.147,Z 412.597,A -85,B 0,C 180,E1 -7387.667,E2 -7387.667} C_VEL
LIN {X 0,Y 474.358,Z 406.145,A -85,B 0,C 180,E1 -7389.38,E2 -7389.38} C_VEL
LIN {X 0,Y 474.783,Z 398.028,A -85,B 0,C 180,E1 -7391.095,E2 -7391.095} C_VEL
LIN {X 0,Y 475.158,Z 389.03,A -85,B 0,C 180,E1 -7392.651,E2 -7392.651} C_VEL
LIN {X 0,Y 475.735,Z 378.853,A -85,B 0,C 180,E1 -7394.108,E2 -7394.108} C_VEL
LIN {X 0,Y 476.313,Z 368.065,A -85,B 0,C 180,E1 -7395.402,E2 -7395.402} C_VEL
LIN {X 0,Y 476.948,Z 356.562,A -85,B 0,C 180,E1 -7396.562,E2 -7396.562} C_VEL
LIN {X 0,Y 477.67,Z 343.417,A -85,B 0,C 180,E1 -7397.666,E2 -7397.666} C_VEL
LIN {X 0,Y 478.233,Z 330.97,A -85,B 0,C 180,E1 -7398.53,E2 -7398.53} C_VEL
LIN {X 0,Y 478.851,Z 316.582,A -85,B 0,C 180,E1 -7399.339,E2 -7399.339} C_VEL
LIN {X 0,Y 479.414,Z 301.265,A -85,B 0,C 180,E1 -7400.003,E2 -7400.003} C_VEL
LIN {X 0,Y 479.81,Z 286.73,A -85,B 0,C 180,E1 -7400.465,E2 -7400.465} C_VEL
LIN {X 0,Y 480.065,Z 269.663,A -85,B 0,C 180,E1 -7400.823,E2 -7400.823} C_VEL
LIN {X 0,Y 482.25,Z 134.507,A -85,B 0,C 180,E1 -7403.116,E2 -7403.116} C_VEL
LIN {X 0,Y 481.409,Z 130.855,A -85,B 0,C 180,E1 -7403.221,E2 -7403.221} C_VEL
LIN {X 0,Y 475.23,Z 114.682,A -85,B 0,C 180,E1 -7403.834,E2 -7403.834} C_VEL
LIN {X 0,Y 474.634,Z 111.989,A -85,B 0,C 180,E1 -7404.32,E2 -7404.32} C_VEL
LIN {X 0,Y 474.639,Z 111.988,A -85,B 0,C 180,E1 -7407.324,E2 -7407.324} C_VEL
LIN {X 0,Y 474.599,Z 111.991,A -85,B 0,C 180,E1 -7410.231,E2 -7410.231} C_VEL
LIN {X 0,Y 474.616,Z 111.99,A -85,B 0,C 180,E1 -7413.223,E2 -7413.223} C_VEL
LIN {X 0,Y 474.585,Z 111.99,A -85,B 0,C 180,E1 -7416.324,E2 -7416.324} C_VEL
LIN {X 0,Y 474.624,Z 111.992,A -85,B 0,C 180,E1 -7419.548,E2 -7419.548} C_VEL
LIN {X 0,Y 474.576,Z 111.994,A -85,B 0,C 180,E1 -7422.939,E2 -7422.939} C_VEL
LIN {X 0,Y 474.603,Z 111.975,A -85,B 0,C 180,E1 -7425.894,E2 -7425.894} C_VEL
LIN {X 0,Y 474.593,Z 111.994,A -85,B 0,C 180,E1 -7429.34,E2 -7429.34} C_VEL
LIN {X 0,Y 474.604,Z 111.988,A -85,B 0,C 180,E1 -7430.329,E2 -7430.329} C_VEL
LIN {X 0,Y 473.969,Z 112.073,A -85,B 0,C 180,E1 -7431.038,E2 -7431.038} C_VEL
LIN {X 0,Y 471.076,Z 112.425,A -85,B 0,C 180,E1 -7432.188,E2 -7432.188} C_VEL
LIN {X 0,Y 468.628,Z 112.729,A -85,B 0,C 180,E1 -7433.115,E2 -7433.115} C_VEL
LIN {X 0,Y 467.612,Z 112.848,A -85,B 0,C 180,E1 -7433.833,E2 -7433.833} C_VEL
LIN {X 0,Y 467.549,Z 112.855,A -85,B 0,C 180,E1 -7434.076,E2 -7434.076} C_VEL
LIN {X 0,Y 467.576,Z 112.868,A -85,B 0,C 180,E1 -7437.241,E2 -7437.241} C_VEL
LIN {X 0,Y 467.537,Z 112.863,A -85,B 0,C 180,E1 -7440.261,E2 -7440.261} C_VEL
LIN {X 0,Y 467.554,Z 112.87,A -85,B 0,C 180,E1 -7443.196,E2 -7443.196} C_VEL
LIN {X 0,Y 467.592,Z 112.858,A -85,B 0,C 180,E1 -7446.47,E2 -7446.47} C_VEL
LIN {X 0,Y 467.614,Z 112.855,A -85,B 0,C 180,E1 -7449.777,E2 -7449.777} C_VEL
LIN {X 0,Y 467.568,Z 112.871,A -85,B 0,C 180,E1 -7452.505,E2 -7452.505} C_VEL
LIN {X 0,Y 467.59,Z 112.864,A -85,B 0,C 180,E1 -7455.196,E2 -7455.196} C_VEL
LIN {X 0,Y 467.66,Z 112.854,A -85,B 0,C 180,E1 -7457.855,E2 -7457.855} C_VEL
LIN {X 0,Y 467.638,Z 112.856,A -85,B 0,C 180,E1 -7461.356,E2 -7461.356} C_VEL
LIN {X 0,Y 467.696,Z 112.852,A -85,B 0,C 180,E1 -7463.962,E2 -7463.962} C_VEL
LIN {X 0,Y 467.814,Z 112.839,A -85,B 0,C 180,E1 -7467.417,E2 -7467.417} C_VEL
LIN {X 0,Y 467.706,Z 112.89,A -85,B 0,C 180,E1 -7468.601,E2 -7468.601} C_VEL
LIN {X 0,Y 470.922,Z 126.715,A -85,B 0,C 180,E1 -7470.769,E2 -7470.769} C_VEL
LIN {X 0,Y 471.732,Z 131.193,A -85,B 0,C 180,E1 -7471.452,E2 -7471.452} C_VEL
LIN {X 0,Y 471.438,Z 142.401,A -85,B 0,C 180,E1 -7473.005,E2 -7473.005} C_VEL
LIN {X 0,Y 475.894,Z 162.991,A -85,B 0,C 180,E1 -7473.576,E2 -7473.576} C_VEL
LIN {X 0,Y 474.115,Z 308.112,A -85,B 0,C 180,E1 -7475.849,E2 -7475.849} C_VEL
LIN {X 0,Y 473.736,Z 323.17,A -85,B 0,C 180,E1 -7476.246,E2 -7476.246} C_VEL
LIN {X 0,Y 473.16,Z 338.329,A -85,B 0,C 180,E1 -7476.824,E2 -7476.824} C_VEL
LIN {X 0,Y 472.536,Z 351.425,A -85,B 0,C 180,E1 -7477.478,E2 -7477.478} C_VEL
LIN {X 0,Y 471.739,Z 365.328,A -85,B 0,C 180,E1 -7478.352,E2 -7478.352} C_VEL
LIN {X 0,Y 470.957,Z 378.071,A -85,B 0,C 180,E1 -7479.34,E2 -7479.34} C_VEL
LIN {X 0,Y 470.061,Z 390.966,A -85,B 0,C 180,E1 -7480.553,E2 -7480.553} C_VEL
LIN {X 0,Y 469.305,Z 402.645,A -85,B 0,C 180,E1 -7481.883,E2 -7481.883} C_VEL
LIN {X 0,Y 468.621,Z 412.536,A -85,B 0,C 180,E1 -7483.221,E2 -7483.221} C_VEL
LIN {X 0,Y 467.985,Z 422.209,A -85,B 0,C 180,E1 -7484.791,E2 -7484.791} C_VEL
LIN {X 0,Y 467.562,Z 429.383,A -85,B 0,C 180,E1 -7486.178,E2 -7486.178} C_VEL
LIN {X 0,Y 467.188,Z 436.949,A -85,B 0,C 180,E1 -7487.962,E2 -7487.962} C_VEL
LIN {X 0,Y 466.904,Z 443.05,A -85,B 0,C 180,E1 -7489.796,E2 -7489.796} C_VEL
LIN {X 0,Y 466.796,Z 446.647,A -85,B 0,C 180,E1 -7491.183,E2 -7491.183} C_VEL
LIN {X 0,Y 466.584,Z 450.256,A -85,B 0,C 180,E1 -7493.056,E2 -7493.056} C_VEL
LIN {X 0,Y 466.489,Z 452.478,A -85,B 0,C 180,E1 -7494.951,E2 -7494.951} C_VEL
LIN {X 0,Y 466.515,Z 453.319,A -85,B 0,C 180,E1 -7496.869,E2 -7496.869} C_VEL
LIN {X 0,Y 466.525,Z 452.745,A -85,B 0,C 180,E1 -7498.82,E2 -7498.82} C_VEL
LIN {X 0,Y 466.586,Z 451.904,A -85,B 0,C 180,E1 -7499.806,E2 -7499.806} C_VEL
LIN {X 0,Y 466.609,Z 450.603,A -85,B 0,C 180,E1 -7500.848,E2 -7500.848} C_VEL
LIN {X 0,Y 466.691,Z 447.626,A -85,B 0,C 180,E1 -7502.507,E2 -7502.507} C_VEL
LIN {X 0,Y 466.901,Z 442.672,A -85,B 0,C 180,E1 -7504.463,E2 -7504.463} C_VEL
LIN {X 0,Y 467.182,Z 436.848,A -85,B 0,C 180,E1 -7506.189,E2 -7506.189} C_VEL
LIN {X 0,Y 467.537,Z 430.048,A -85,B 0,C 180,E1 -7507.803,E2 -7507.803} C_VEL
LIN {X 0,Y 468.019,Z 421.966,A -85,B 0,C 180,E1 -7509.379,E2 -7509.379} C_VEL
LIN {X 0,Y 468.572,Z 413.703,A -85,B 0,C 180,E1 -7510.726,E2 -7510.726} C_VEL
LIN {X 0,Y 469.272,Z 403.664,A -85,B 0,C 180,E1 -7512.113,E2 -7512.113} C_VEL
LIN {X 0,Y 470.032,Z 392.061,A -85,B 0,C 180,E1 -7513.456,E2 -7513.456} C_VEL
LIN {X 0,Y 470.821,Z 380.7,A -85,B 0,C 180,E1 -7514.554,E2 -7514.554} C_VEL
LIN {X 0,Y 471.604,Z 368.509,A -85,B 0,C 180,E1 -7515.54,E2 -7515.54} C_VEL
LIN {X 0,Y 472.463,Z 354.191,A -85,B 0,C 180,E1 -7516.483,E2 -7516.483} C_VEL
LIN {X 0,Y 473.102,Z 340.613,A -85,B 0,C 180,E1 -7517.195,E2 -7517.195} C_VEL
LIN {X 0,Y 473.733,Z 325.519,A -85,B 0,C 180,E1 -7517.795,E2 -7517.795} C_VEL
LIN {X 0,Y 474.176,Z 311.304,A -85,B 0,C 180,E1 -7518.195,E2 -7518.195} C_VEL
LIN {X 0,Y 474.464,Z 288.06,A -85,B 0,C 180,E1 -7518.6,E2 -7518.6} C_VEL
LIN {X 0,Y 475.971,Z 158.129,A -85,B 0,C 180,E1 -7520.635,E2 -7520.635} C_VEL
LIN {X 0,Y 472.761,Z 140.715,A -85,B 0,C 180,E1 -7521.114,E2 -7521.114} C_VEL
LIN {X 0,Y 472.903,Z 132.941,A -85,B 0,C 180,E1 -7521.967,E2 -7521.967} C_VEL
LIN {X 0,Y 468.733,Z 117.016,A -85,B 0,C 180,E1 -7523.976,E2 -7523.976} C_VEL
LIN {X 0,Y 467.587,Z 112.868,A -85,B 0,C 180,E1 -7524.527,E2 -7524.527} C_VEL
LIN {X 0,Y 467.584,Z 112.867,A -85,B 0,C 180,E1 -7527.321,E2 -7527.321} C_VEL
LIN {X 0,Y 467.572,Z 112.863,A -85,B 0,C 180,E1 -7530.667,E2 -7530.667} C_VEL
LIN {X 0,Y 467.619,Z 112.863,A -85,B 0,C 180,E1 -7533.2,E2 -7533.2} C_VEL
LIN {X 0,Y 467.599,Z 112.866,A -85,B 0,C 180,E1 -7535.644,E2 -7535.644} C_VEL
LIN {X 0,Y 467.998,Z 114.447,A -85,B 0,C 180,E1 -7535.876,E2 -7535.876} C_VEL
LIN {X 0,Y 475.718,Z 134.089,A -85,B 0,C 180,E1 -7536.635,E2 -7536.635} C_VEL
LIN {X 0,Y 473.186,Z 282.051,A -85,B 0,C 180,E1 -7539.232,E2 -7539.232} C_VEL
LIN {X 0,Y 472.831,Z 297.106,A -85,B 0,C 180,E1 -7539.664,E2 -7539.664} C_VEL
LIN {X 0,Y 472.295,Z 312.136,A -85,B 0,C 180,E1 -7540.269,E2 -7540.269} C_VEL
LIN {X 0,Y 471.681,Z 325.748,A -85,B 0,C 180,E1 -7540.977,E2 -7540.977} C_VEL
LIN {X 0,Y 471.016,Z 339.2,A -85,B 0,C 180,E1 -7541.852,E2 -7541.852} C_VEL
LIN {X 0,Y 470.321,Z 352.691,A -85,B 0,C 180,E1 -7542.926,E2 -7542.926} C_VEL
LIN {X 0,Y 469.616,Z 365.347,A -85,B 0,C 180,E1 -7544.15,E2 -7544.15} C_VEL
LIN {X 0,Y 468.966,Z 376.664,A -85,B 0,C 180,E1 -7545.462,E2 -7545.462} C_VEL
LIN {X 0,Y 468.374,Z 386.18,A -85,B 0,C 180,E1 -7546.772,E2 -7546.772} C_VEL
LIN {X 0,Y 467.913,Z 395.504,A -85,B 0,C 180,E1 -7548.301,E2 -7548.301} C_VEL
LIN {X 0,Y 467.468,Z 403.222,A -85,B 0,C 180,E1 -7549.825,E2 -7549.825} C_VEL
LIN {X 0,Y 467.233,Z 409.59,A -85,B 0,C 180,E1 -7551.349,E2 -7551.349} C_VEL
LIN {X 0,Y 466.974,Z 415.418,A -85,B 0,C 180,E1 -7553.084,E2 -7553.084} C_VEL
LIN {X 0,Y 466.897,Z 418.888,A -85,B 0,C 180,E1 -7554.385,E2 -7554.385} C_VEL
LIN {X 0,Y 466.806,Z 421.554,A -85,B 0,C 180,E1 -7555.683,E2 -7555.683} C_VEL
LIN {X 0,Y 466.797,Z 424.069,A -85,B 0,C 180,E1 -7557.411,E2 -7557.411} C_VEL
LIN {X 0,Y 466.63,Z 425.402,A -85,B 0,C 180,E1 -7559.137,E2 -7559.137} C_VEL
LIN {X 0,Y 466.631,Z 425.506,A -85,B 0,C 180,E1 -7560.863,E2 -7560.863} C_VEL
LIN {X 0,Y 466.83,Z 424.414,A -85,B 0,C 180,E1 -7562.588,E2 -7562.588} C_VEL
LIN {X 0,Y 466.863,Z 422.139,A -85,B 0,C 180,E1 -7564.316,E2 -7564.316} C_VEL
LIN {X 0,Y 467.017,Z 418.61,A -85,B 0,C 180,E1 -7566.047,E2 -7566.047} C_VEL
LIN {X 0,Y 467.161,Z 413.757,A -85,B 0,C 180,E1 -7567.781,E2 -7567.781} C_VEL
LIN {X 0,Y 467.443,Z 407.44,A -85,B 0,C 180,E1 -7569.519,E2 -7569.519} C_VEL
LIN {X 0,Y 467.857,Z 399.448,A -85,B 0,C 180,E1 -7571.261,E2 -7571.261} C_VEL
LIN {X 0,Y 468.339,Z 390.552,A -85,B 0,C 180,E1 -7572.841,E2 -7572.841} C_VEL
LIN {X 0,Y 469.009,Z 380.506,A -85,B 0,C 180,E1 -7574.315,E2 -7574.315} C_VEL
LIN {X 0,Y 469.633,Z 369.818,A -85,B 0,C 180,E1 -7575.626,E2 -7575.626} C_VEL
LIN {X 0,Y 470.316,Z 358.162,A -85,B 0,C 180,E1 -7576.828,E2 -7576.828} C_VEL
LIN {X 0,Y 471.012,Z 345.397,A -85,B 0,C 180,E1 -7577.923,E2 -7577.923} C_VEL
LIN {X 0,Y 471.789,Z 331.36,A -85,B 0,C 180,E1 -7578.905,E2 -7578.905} C_VEL
LIN {X 0,Y 472.357,Z 317.801,A -85,B 0,C 180,E1 -7579.671,E2 -7579.671} C_VEL
LIN {X 0,Y 472.941,Z 302.747,A -85,B 0,C 180,E1 -7580.33,E2 -7580.33} C_VEL
LIN {X 0,Y 473.359,Z 287.326,A -85,B 0,C 180,E1 -7580.823,E2 -7580.823} C_VEL
LIN {X 0,Y 473.749,Z 264.871,A -85,B 0,C 180,E1 -7581.284,E2 -7581.284} C_VEL
LIN {X 0,Y 475.839,Z 179.153,A -85,B 0,C 180,E1 -7582.925,E2 -7582.925} C_VEL
LIN {X 0,Y 477.016,Z 136.846,A -85,B 0,C 180,E1 -7583.793,E2 -7583.793} C_VEL
LIN {X 0,Y 471.473,Z 124.639,A -85,B 0,C 180,E1 -7584.477,E2 -7584.477} C_VEL
LIN {X 0,Y 469.821,Z 121.428,A -85,B 0,C 180,E1 -7584.693,E2 -7584.693} C_VEL
LIN {X 0,Y 467.563,Z 112.872,A -85,B 0,C 180,E1 -7586.803,E2 -7586.803} C_VEL
LIN {X 0,Y 467.542,Z 112.874,A -85,B 0,C 180,E1 -7589.739,E2 -7589.739} C_VEL
LIN {X 0,Y 467.573,Z 112.868,A -85,B 0,C 180,E1 -7592.759,E2 -7592.759} C_VEL
LIN {X 0,Y 467.55,Z 112.871,A -85,B 0,C 180,E1 -7595.89,E2 -7595.89} C_VEL
LIN {X 0,Y 467.552,Z 112.872,A -85,B 0,C 180,E1 -7599.147,E2 -7599.147} C_VEL
LIN {X 0,Y 467.558,Z 112.871,A -85,B 0,C 180,E1 -7601.405,E2 -7601.405} C_VEL
LIN {X 0,Y 467.564,Z 112.87,A -85,B 0,C 180,E1 -7605.052,E2 -7605.052} C_VEL
LIN {X 0,Y 467.559,Z 112.871,A -85,B 0,C 180,E1 -7608.726,E2 -7608.726} C_VEL
LIN {X 0,Y 467.559,Z 112.869,A -85,B 0,C 180,E1 -7611.955,E2 -7611.955} C_VEL
LIN {X 0,Y 467.553,Z 112.873,A -85,B 0,C 180,E1 -7615.166,E2 -7615.166} C_VEL
LIN {X 0,Y 467.559,Z 112.926,A -85,B 0,C 180,E1 -7617.45,E2 -7617.45} C_VEL
LIN {X 0,Y 470.758,Z 124.137,A -85,B 0,C 180,E1 -7619.701,E2 -7619.701} C_VEL
LIN {X 0,Y 472.806,Z 132.869,A -85,B 0,C 180,E1 -7621.283,E2 -7621.283} C_VEL
LIN {X 0,Y 472.96,Z 136.402,A -85,B 0,C 180,E1 -7621.849,E2 -7621.849} C_VEL
LIN {X 0,Y 471.672,Z 153.837,A -85,B 0,C 180,E1 -7624.399,E2 -7624.399} C_VEL
LIN {X 0,Y 471.224,Z 161.007,A -85,B 0,C 180,E1 -7625.422,E2 -7625.422} C_VEL
LIN {X 0,Y 474.768,Z 180.278,A -85,B 0,C 180,E1 -7626.105,E2 -7626.105} C_VEL
LIN {X 0,Y 476.162,Z 191,A -85,B 0,C 180,E1 -7626.43,E2 -7626.43} C_VEL
LIN {X 0,Y 473.921,Z 284.293,A -85,B 0,C 180,E1 -7628.239,E2 -7628.239} C_VEL
LIN {X 0,Y 473.014,Z 331.076,A -85,B 0,C 180,E1 -7629.109,E2 -7629.109} C_VEL
LIN {X 0,Y 472.33,Z 347.404,A -85,B 0,C 180,E1 -7629.581,E2 -7629.581} C_VEL
LIN {X 0,Y 471.81,Z 363.699,A -85,B 0,C 180,E1 -7630.191,E2 -7630.191} C_VEL
LIN {X 0,Y 471.196,Z 376.85,A -85,B 0,C 180,E1 -7630.844,E2 -7630.844} C_VEL
LIN {X 0,Y 470.564,Z 390.787,A -85,B 0,C 180,E1 -7631.721,E2 -7631.721} C_VEL
LIN {X 0,Y 469.803,Z 403.637,A -85,B 0,C 180,E1 -7632.715,E2 -7632.715} C_VEL
LIN {X 0,Y 469.169,Z 414.845,A -85,B 0,C 180,E1 -7633.758,E2 -7633.758} C_VEL
LIN {X 0,Y 468.531,Z 426.098,A -85,B 0,C 180,E1 -7635.004,E2 -7635.004} C_VEL
LIN {X 0,Y 467.995,Z 436.094,A -85,B 0,C 180,E1 -7636.319,E2 -7636.319} C_VEL
LIN {X 0,Y 467.449,Z 445.826,A -85,B 0,C 180,E1 -7637.849,E2 -7637.849} C_VEL
LIN {X 0,Y 467.193,Z 453.904,A -85,B 0,C 180,E1 -7639.381,E2 -7639.381} C_VEL
LIN {X 0,Y 466.902,Z 460.587,A -85,B 0,C 180,E1 -7640.906,E2 -7640.906} C_VEL
LIN {X 0,Y 466.807,Z 466.697,A -85,B 0,C 180,E1 -7642.648,E2 -7642.648} C_VEL
LIN {X 0,Y 466.748,Z 470.284,A -85,B 0,C 180,E1 -7643.95,E2 -7643.95} C_VEL
LIN {X 0,Y 466.651,Z 473.946,A -85,B 0,C 180,E1 -7645.681,E2 -7645.681} C_VEL
LIN {X 0,Y 466.705,Z 476.363,A -85,B 0,C 180,E1 -7647.411,E2 -7647.411} C_VEL
LIN {X 0,Y 466.62,Z 477.566,A -85,B 0,C 180,E1 -7649.137,E2 -7649.137} C_VEL
LIN {X 0,Y 466.62,Z 477.616,A -85,B 0,C 180,E1 -7650.863,E2 -7650.863} C_VEL
LIN {X 0,Y 466.695,Z 476.427,A -85,B 0,C 180,E1 -7652.589,E2 -7652.589} C_VEL
LIN {X 0,Y 466.645,Z 473.991,A -85,B 0,C 180,E1 -7654.319,E2 -7654.319} C_VEL
LIN {X 0,Y 466.748,Z 470.323,A -85,B 0,C 180,E1 -7656.05,E2 -7656.05} C_VEL
LIN {X 0,Y 466.81,Z 465.324,A -85,B 0,C 180,E1 -7657.787,E2 -7657.787} C_VEL
LIN {X 0,Y 466.93,Z 458.851,A -85,B 0,C 180,E1 -7659.53,E2 -7659.53} C_VEL
LIN {X 0,Y 467.242,Z 451.819,A -85,B 0,C 180,E1 -7661.057,E2 -7661.057} C_VEL
LIN {X 0,Y 467.586,Z 443.572,A -85,B 0,C 180,E1 -7662.544,E2 -7662.544} C_VEL
LIN {X 0,Y 468.018,Z 434.613,A -85,B 0,C 180,E1 -7663.902,E2 -7663.902} C_VEL
LIN {X 0,Y 468.644,Z 424.332,A -85,B 0,C 180,E1 -7665.215,E2 -7665.215} C_VEL
LIN {X 0,Y 469.317,Z 411.962,A -85,B 0,C 180,E1 -7666.53,E2 -7666.53} C_VEL
LIN {X 0,Y 469.986,Z 399.52,A -85,B 0,C 180,E1 -7667.627,E2 -7667.627} C_VEL
LIN {X 0,Y 470.742,Z 385.798,A -85,B 0,C 180,E1 -7668.61,E2 -7668.61} C_VEL
LIN {X 0,Y 471.596,Z 369.755,A -85,B 0,C 180,E1 -7669.535,E2 -7669.535} C_VEL
LIN {X 0,Y 472.259,Z 354.188,A -85,B 0,C 180,E1 -7670.231,E2 -7670.231} C_VEL
LIN {X 0,Y 472.826,Z 338.766,A -85,B 0,C 180,E1 -7670.732,E2 -7670.732} C_VEL
LIN {X 0,Y 473.178,Z 322.307,A -85,B 0,C 180,E1 -7671.083,E2 -7671.083} C_VEL
LIN {X 0,Y 475.486,Z 187.13,A -85,B 0,C 180,E1 -7673.429,E2 -7673.429} C_VEL
LIN {X 0,Y 473.665,Z 172.835,A -85,B 0,C 180,E1 -7673.835,E2 -7673.835} C_VEL
LIN {X 0,Y 472.304,Z 162.252,A -85,B 0,C 180,E1 -7674.184,E2 -7674.184} C_VEL
LIN {X 0,Y 473.657,Z 135.03,A -85,B 0,C 180,E1 -7677.094,E2 -7677.094} C_VEL
LIN {X 0,Y 467.6,Z 112.866,A -85,B 0,C 180,E1 -7679.952,E2 -7679.952} C_VEL
LIN {X 0,Y 467.572,Z 112.868,A -85,B 0,C 180,E1 -7682.759,E2 -7682.759} C_VEL
LIN {X 0,Y 467.549,Z 112.869,A -85,B 0,C 180,E1 -7685.89,E2 -7685.89} C_VEL
LIN {X 0,Y 467.551,Z 112.872,A -85,B 0,C 180,E1 -7689.148,E2 -7689.148} C_VEL
LIN {X 0,Y 467.557,Z 112.868,A -85,B 0,C 180,E1 -7691.405,E2 -7691.405} C_VEL
LIN {X 0,Y 467.564,Z 112.867,A -85,B 0,C 180,E1 -7695.053,E2 -7695.053} C_VEL
LIN {X 0,Y 467.559,Z 112.869,A -85,B 0,C 180,E1 -7698.726,E2 -7698.726} C_VEL
LIN {X 0,Y 467.56,Z 112.869,A -85,B 0,C 180,E1 -7701.955,E2 -7701.955} C_VEL
LIN {X 0,Y 467.555,Z 112.869,A -85,B 0,C 180,E1 -7705.167,E2 -7705.167} C_VEL
LIN {X 0,Y 467.577,Z 112.869,A -85,B 0,C 180,E1 -7708.26,E2 -7708.26} C_VEL
LIN {X 0,Y 467.545,Z 112.872,A -85,B 0,C 180,E1 -7711.249,E2 -7711.249} C_VEL
LIN {X 0,Y 467.567,Z 112.937,A -85,B 0,C 180,E1 -7714.348,E2 -7714.348} C_VEL
LIN {X 0,Y 469.493,Z 119.217,A -85,B 0,C 180,E1 -7715.39,E2 -7715.39} C_VEL
LIN {X 0,Y 475.937,Z 133.241,A -85,B 0,C 180,E1 -7716.19,E2 -7716.19} C_VEL
LIN {X 0,Y 476.97,Z 136.048,A -85,B 0,C 180,E1 -7716.324,E2 -7716.324} C_VEL
LIN {X 0,Y 474.487,Z 226.823,A -85,B 0,C 180,E1 -7718.124,E2 -7718.124} C_VEL
LIN {X 0,Y 473.352,Z 284.62,A -85,B 0,C 180,E1 -7719.217,E2 -7719.217} C_VEL
LIN {X 0,Y 472.884,Z 301.059,A -85,B 0,C 180,E1 -7719.711,E2 -7719.711} C_VEL
LIN {X 0,Y 472.332,Z 316.706,A -85,B 0,C 180,E1 -7720.384,E2 -7720.384} C_VEL
LIN {X 0,Y 471.736,Z 331.303,A -85,B 0,C 180,E1 -7721.206,E2 -7721.206} C_VEL
LIN {X 0,Y 470.993,Z 345.318,A -85,B 0,C 180,E1 -7722.188,E2 -7722.188} C_VEL
